	// Row 2: Time (seconds)
	GVL_HMI.aSolventAndTimesRows[2].Rinse1 := DWORD_TO_INT(TIME_TO_DWORD(GVL_Recipe.stCurrentRecipe.stSolventsTimes.aTime[1]) / 1000); // TIME in seconds
	GVL_HMI.aSolventAndTimesRows[2].Rinse2 := DWORD_TO_INT(TIME_TO_DWORD(GVL_Recipe.stCurrentRecipe.stSolventsTimes.aTime[2]) / 1000); // TIME in seconds
	GVL_HMI.aSolventAndTimesRows[2].Wash1  := DWORD_TO_INT(TIME_TO_DWORD(GVL_Recipe.stCurrentRecipe.stSolventsTimes.aTime[3]) / 1000); // TIME in seconds
	GVL_HMI.aSolventAndTimesRows[2].Wash2  := DWORD_TO_INT(TIME_TO_DWORD(GVL_Recipe.stCurrentRecipe.stSolventsTimes.aTime[4]) / 1000); // TIME in seconds
	
	// Row 3: Velocity
	GVL_HMI.aSolventAndTimesRows[3].Rinse1 := GVL_Recipe.stCurrentRecipe.stSolventsTimes.aVelocity[1];
	GVL_HMI.aSolventAndTimesRows[3].Rinse2 := GVL_Recipe.stCurrentRecipe.stSolventsTimes.aVelocity[2];
	GVL_HMI.aSolventAndTimesRows[3].Wash1  := GVL_Recipe.stCurrentRecipe.stSolventsTimes.aVelocity[3];
	GVL_HMI.aSolventAndTimesRows[3].Wash2  := GVL_Recipe.stCurrentRecipe.stSolventsTimes.aVelocity[4];
	
	//Volumes Datagrid
	// 1:Rinse1, 2:Rinse2, 3:Wash1, 4:Wash2
    GVL_HMI.aVolumeRows[1].Rinse1 := GVL_Recipe.stCurrentRecipe.stVolumes.aT_IC_Volume[1];
    GVL_HMI.aVolumeRows[1].Rinse2 := GVL_Recipe.stCurrentRecipe.stVolumes.aT_IC_Volume[2];
    GVL_HMI.aVolumeRows[1].Wash1  := GVL_Recipe.stCurrentRecipe.stVolumes.aT_IC_Volume[3];
    GVL_HMI.aVolumeRows[1].Wash2  := GVL_Recipe.stCurrentRecipe.stVolumes.aT_IC_Volume[4];

    GVL_HMI.aVolumeRows[2].Rinse1 := GVL_Recipe.stCurrentRecipe.stVolumes.aS0_Volume[1];
    GVL_HMI.aVolumeRows[2].Rinse2 := GVL_Recipe.stCurrentRecipe.stVolumes.aS0_Volume[2];
    GVL_HMI.aVolumeRows[2].Wash1  := GVL_Recipe.stCurrentRecipe.stVolumes.aS0_Volume[3];
    GVL_HMI.aVolumeRows[2].Wash2  := GVL_Recipe.stCurrentRecipe.stVolumes.aS0_Volume[4];

    GVL_HMI.aVolumeRows[3].Rinse1 := GVL_Recipe.stCurrentRecipe.stVolumes.aS1_Volume[1];
    GVL_HMI.aVolumeRows[3].Rinse2 := GVL_Recipe.stCurrentRecipe.stVolumes.aS1_Volume[2];
   	GVL_HMI.aVolumeRows[3].Wash1  := GVL_Recipe.stCurrentRecipe.stVolumes.aS1_Volume[3];
    GVL_HMI.aVolumeRows[3].Wash2  := GVL_Recipe.stCurrentRecipe.stVolumes.aS1_Volume[4];
	
	GVL_HMI.aVolumeRows[4].Rinse1 := GVL_Recipe.stCurrentRecipe.stVolumes.aS2_Volume[1];
    GVL_HMI.aVolumeRows[4].Rinse2 := GVL_Recipe.stCurrentRecipe.stVolumes.aS2_Volume[2];
   	GVL_HMI.aVolumeRows[4].Wash1  := GVL_Recipe.stCurrentRecipe.stVolumes.aS2_Volume[3];
    GVL_HMI.aVolumeRows[4].Wash2  := GVL_Recipe.stCurrentRecipe.stVolumes.aS2_Volume[4];
	
	GVL_HMI.aVolumeRows[5].Rinse1 := GVL_Recipe.stCurrentRecipe.stVolumes.aS3_Volume[1];
    GVL_HMI.aVolumeRows[5].Rinse2 := GVL_Recipe.stCurrentRecipe.stVolumes.aS3_Volume[2];
   	GVL_HMI.aVolumeRows[5].Wash1  := GVL_Recipe.stCurrentRecipe.stVolumes.aS3_Volume[3];
    GVL_HMI.aVolumeRows[5].Wash2  := GVL_Recipe.stCurrentRecipe.stVolumes.aS3_Volume[4];
	
	GVL_HMI.aVolumeRows[6].Rinse1 := GVL_Recipe.stCurrentRecipe.stVolumes.aS4_Volume[1];
    GVL_HMI.aVolumeRows[6].Rinse2 := GVL_Recipe.stCurrentRecipe.stVolumes.aS4_Volume[2];
   	GVL_HMI.aVolumeRows[6].Wash1  := GVL_Recipe.stCurrentRecipe.stVolumes.aS4_Volume[3];
    GVL_HMI.aVolumeRows[6].Wash2  := GVL_Recipe.stCurrentRecipe.stVolumes.aS4_Volume[4];
	
	GVL_HMI.aVolumeRows[7].Rinse1 := GVL_Recipe.stCurrentRecipe.stVolumes.aS5_Volume[1];
    GVL_HMI.aVolumeRows[7].Rinse2 := GVL_Recipe.stCurrentRecipe.stVolumes.aS5_Volume[2];
   	GVL_HMI.aVolumeRows[7].Wash1  := GVL_Recipe.stCurrentRecipe.stVolumes.aS5_Volume[3];
    GVL_HMI.aVolumeRows[7].Wash2  := GVL_Recipe.stCurrentRecipe.stVolumes.aS5_Volume[4];
	
	GVL_HMI.aVolumeRows[8].Rinse1 := GVL_Recipe.stCurrentRecipe.stVolumes.aS6_Volume[1];
    GVL_HMI.aVolumeRows[8].Rinse2 := GVL_Recipe.stCurrentRecipe.stVolumes.aS6_Volume[2];
   	GVL_HMI.aVolumeRows[8].Wash1  := GVL_Recipe.stCurrentRecipe.stVolumes.aS6_Volume[3];
    GVL_HMI.aVolumeRows[8].Wash2  := GVL_Recipe.stCurrentRecipe.stVolumes.aS6_Volume[4];
	
	GVL_HMI.aVolumeRows[9].Rinse1 := GVL_Recipe.stCurrentRecipe.stVolumes.aS7_Volume[1];
    GVL_HMI.aVolumeRows[9].Rinse2 := GVL_Recipe.stCurrentRecipe.stVolumes.aS7_Volume[2];
   	GVL_HMI.aVolumeRows[9].Wash1  := GVL_Recipe.stCurrentRecipe.stVolumes.aS7_Volume[3];
    GVL_HMI.aVolumeRows[9].Wash2  := GVL_Recipe.stCurrentRecipe.stVolumes.aS7_Volume[4];

    GVL_HMI.aVolumeRows[10].Rinse1 := GVL_Recipe.stCurrentRecipe.stVolumes.aF_Volume[1];
    GVL_HMI.aVolumeRows[10].Rinse2 := GVL_Recipe.stCurrentRecipe.stVolumes.aF_Volume[2];
    GVL_HMI.aVolumeRows[10].Wash1  := GVL_Recipe.stCurrentRecipe.stVolumes.aF_Volume[3];
    GVL_HMI.aVolumeRows[10].Wash2  := GVL_Recipe.stCurrentRecipe.stVolumes.aF_Volume[4];
	
	//Other Params datagrid
	GVL_HMI.aOtherParamsRows[1].Value     := TIME_TO_DWORD(GVL_Recipe.stCurrentRecipe.stOtherParams.tSoakTime) / 1000.0; // Soak Time
	GVL_HMI.aOtherParamsRows[2].Value     := TIME_TO_DWORD(GVL_Recipe.stCurrentRecipe.stOtherParams.tAgitate1Time) / 1000.0; // Agitate 1 Time
	GVL_HMI.aOtherParamsRows[3].Value     := TIME_TO_DWORD(GVL_Recipe.stCurrentRecipe.stOtherParams.tAgitate2Time) / 1000.0; // Agitate 2 Time
	GVL_HMI.aOtherParamsRows[4].Value     := GVL_Recipe.stCurrentRecipe.stOtherParams.iVialsToFill; // Vials to Fill
	GVL_HMI.aOtherParamsRows[5].Value     := GVL_Recipe.stCurrentRecipe.stOtherParams.rVialPrimeVol; // Vial Prime Vol
	GVL_HMI.aOtherParamsRows[6].Value     := GVL_Recipe.stCurrentRecipe.stOtherParams.rVial1FillVol; // Vial 1 Fill Vol
	GVL_HMI.aOtherParamsRows[7].Value     := GVL_Recipe.stCurrentRecipe.stOtherParams.rVials2_4FillVol; // Vials 2-4 Fill Vol
	GVL_HMI.aOtherParamsRows[8].Value     := TIME_TO_DWORD(GVL_Recipe.stCurrentRecipe.stOtherParams.tAirDryTime) / 1000.0; // Air Dry Time
	
	iStep := 100;

90:
    fbFileClose(sNetId := '', hFile := hFile, bExecute := TRUE);
    iStep := 100;
	
100:
    bBusy := FALSE;
    bDone := NOT bError;
    IF NOT bExecute THEN
        iStep := 0;
    END_IF
END_CASE

END_FUNCTION_BLOCK

// ---- POUs/4. RecipeHandle/FB_ListRecipeFiles.TcPOU
// FB_ListRecipeFiles: Scans the recipe folder and fills GVL_Recipe.aAvailableFiles with metadata from JSON files
FUNCTION_BLOCK FB_ListRecipeFiles
VAR_INPUT
	bExecute : BOOL; // Start the file listing process
END_VAR
VAR_OUTPUT
	bBusy       : BOOL; // Indicates the block is busy
    bError      : BOOL; // Indicates an error occurred
    nErrId      : UDINT; // Error code if any
	bDone   	: BOOL;

END_VAR
VAR
	fbEnumFiles     : FB_EnumFindFileList;
    fbFileTime      : FB_FileTime64ToTzSpecificLocalTime;
    fbHeaderHandler : FB_RecipeHeaderHandler;

    aFindBuffer     : ARRAY[0..49] OF ST_FindFileEntry;
    nFoundFiles     : UDINT;
    iFileIndex      : INT;
    iStep           : INT;
    bExecutePrev    : BOOL;
    bStart          : BOOL;
    bHeaderHandlerReset : BOOL;
    bHeaderHandlerExecute : BOOL;
	
	i : INT;
	
END_VAR

bStart := NOT bExecutePrev AND bExecute;
bExecutePrev := bExecute;

IF NOT bExecute THEN
	bBusy := FALSE;
  	bDone := FALSE;
	bError := FALSE;
	nErrId := 0;
END_IF

CASE iStep OF

0:
    IF bStart THEN
        bBusy := TRUE;
        bDone := FALSE;
        bError := FALSE;
        nErrId := 0;
        iFileIndex := 0;
        bHeaderHandlerReset := FALSE;
        bHeaderHandlerExecute := FALSE;

        fbEnumFiles(
            sNetId := '',
            sPathName := 'C:/TwinCAT/Recipes/*.json',
            eCmd := eEnumCmd_First,
            pFindList := ADR(aFindBuffer),
            cbFindList := SIZEOF(aFindBuffer),
            bExecute := TRUE
        );

        iStep := 10;
    END_IF

10:
    fbEnumFiles(bExecute := FALSE);
    IF NOT fbEnumFiles.bBusy THEN
        IF fbEnumFiles.bError THEN
            bError := TRUE;
            nErrId := fbEnumFiles.nErrId;
            iStep := 100;
        ELSE
            nFoundFiles := fbEnumFiles.nFindFiles;
            IF nFoundFiles > 0 THEN
                iStep := 20;
            ELSE
                bDone := TRUE;
                iStep := 100;
            END_IF
        END_IF
    END_IF

// 20 - Processa arquivo iFileIndex
20:
    IF iFileIndex < TO_INT(nFoundFiles) AND iFileIndex <= 49 THEN
        // Preenche campos básicos do arquivo
        GVL_HMI.aAvailableFiles[iFileIndex].sFileName := aFindBuffer[iFileIndex].sFileName;
        fbFileTime(
            in := FILETIME_TO_FILETIME64(aFindBuffer[iFileIndex].lastWriteTime),
            tzInfo := WEST_EUROPE_TZI
        );
        GVL_HMI.aAvailableFiles[iFileIndex].dtLastModified := FILETIME64_TO_DT(fbFileTime.out);

        // Vai para o step de reset do FB_HeaderHandler
        iStep := 21;
    ELSE
        bDone := TRUE;
        iStep := 100;
    END_IF

// 21 - Reset do FB_HeaderHandler (chamada com bExecute := FALSE por um ciclo)
21:
    fbHeaderHandler(bExecute := FALSE);
    IF NOT fbHeaderHandler.bBusy AND NOT fbHeaderHandler.bDone THEN
        iStep := 22;
    END_IF

// 22 - Chama o FB_HeaderHandler para ler o header do arquivo atual
22:
    fbHeaderHandler(
        sFileName := CONCAT('C:/TwinCAT/Recipes/', aFindBuffer[iFileIndex].sFileName),
        iTargetIndex := iFileIndex,
        bExecute := TRUE
    );
    IF NOT fbHeaderHandler.bBusy THEN
        IF fbHeaderHandler.bError THEN
            bError := TRUE;
            nErrId := fbHeaderHandler.nErrId;
            iStep := 100;
        ELSIF fbHeaderHandler.bDone THEN
            iStep := 23;
        END_IF
    END_IF

23: // Dummy step — aguarda 1 ciclo antes de liberar novo arquivo
    fbHeaderHandler(bExecute := FALSE);
    iFileIndex := iFileIndex + 1;
    iStep := 20;

100:
    bBusy := FALSE;
    IF NOT bExecute THEN
        iStep := 0;
    END_IF
END_CASE

END_FUNCTION_BLOCK

// ---- POUs/4. RecipeHandle/FB_RecipeHeaderHandler.TcPOU
// FB_RecipeHeaderHandler: Extracts metadata from a recipe JSON file and fills one entry in GVL_Recipe.aAvailableFiles
FUNCTION_BLOCK FB_RecipeHeaderHandler
VAR_INPUT
	sFileName       : STRING(255);
    iTargetIndex    : INT; // Index to write into array GVL_Recipe.aAvailableFiles
    bExecute        : BOOL;
END_VAR
VAR_OUTPUT
	bBusy  : BOOL;
    bError : BOOL;
    bDone  : BOOL;
    nErrId : UDINT;
END_VAR
VAR
	iStep         : INT;
    hFile         : UINT;
    sBuffer       : STRING(8192);
    fbFileOpen    : FB_FileOpen;
    fbFileRead    : FB_FileRead;
    fbFileClose   : FB_FileClose;
    fbJson        : FB_JsonDomParser;
    jsonDoc       : SJsonValue;
    jsonProp      : SJsonValue;
	nBytesRead    : UDINT;
	bExecutePrev  : BOOL; 
    bStart        : BOOL;
	bWait1Cycle	  : BOOL := FALSE;
	iCount		  : UINT := 0;
	iDummyTimer	  : INT := 0;
END_VAR

bStart := bExecute AND NOT bExecutePrev;
bExecutePrev := bExecute;

IF NOT bExecute THEN
	bBusy := FALSE;
    bDone := FALSE;
    bError := FALSE;

	sBuffer := '';
	jsonDoc := 0;
	jsonProp := 0;
	hFile := 0;
	bExecutePrev := FALSE;	
END_IF

CASE iStep OF

0:
     IF bExecute AND NOT bBusy THEN
        bBusy := TRUE;
        bDone := FALSE;
        bError := FALSE;
        nErrId := 0;
        iCount := 0;
        // Reset interno total
        sBuffer := '';
        jsonDoc := 0;
        jsonProp := 0;
        hFile := 0;
        iStep := 5;
    END_IF
	
5:
	fbFileOpen(
            sNetId := '',
            sPathName := sFileName,
            nMode := FOPEN_MODEREAD OR FOPEN_MODETEXT,
            bExecute := TRUE,
			hFile => hFile
	);
	IF NOT fbFileOpen.bBusy AND NOT fbFileOpen.bError THEN
		iStep := 10;
	END_IF

10:
    fbFileOpen(
        sNetId := '',
        sPathName := sFileName,
        nMode := FOPEN_MODEREAD OR FOPEN_MODETEXT,
        bExecute := FALSE
    );
    IF NOT fbFileOpen.bBusy THEN
        IF fbFileOpen.bError THEN
            bError := TRUE;
            nErrId := fbFileOpen.nErrId;
            iStep := 100;
        ELSE
            hFile := fbFileOpen.hFile;
            fbFileRead(
                sNetId := '',
                hFile := hFile,
                pReadBuff := ADR(sBuffer),
                cbReadLen := SIZEOF(sBuffer),
                bExecute := TRUE
            );
            iStep := 20;
        END_IF
    END_IF

20:
    fbFileRead(
        sNetId := '',
        hFile := hFile,
        pReadBuff := ADR(sBuffer),
        cbReadLen := SIZEOF(sBuffer),
        bExecute := FALSE,
        cbRead => nBytesRead 
    );
    IF NOT fbFileRead.bBusy THEN
        IF fbFileRead.bError THEN
            bError := TRUE;
            nErrId := fbFileRead.nErrId;
            iStep := 100;
        ELSE
            // Clear the buffer
            IF nBytesRead < SIZEOF(sBuffer) THEN
    			sBuffer[nBytesRead] := 0; 
			END_IF

            fbFileClose(
                sNetId := '',
                hFile := hFile,
                bExecute := TRUE
            );
            iStep := 30;
        END_IF
    END_IF


30:
    fbFileClose(
        sNetId := '',
        hFile := hFile,
        bExecute := FALSE
    );
    IF NOT fbFileClose.bBusy THEN
        IF fbFileClose.bError THEN
            bError := TRUE;
            nErrId := fbFileClose.nErrId;
            iStep := 100;
        ELSE
            iStep := 31;
        END_IF
    END_IF

31: // Dummy step: espera um ciclo para garantir flush/GC do Windows
	fbFileClose( sNetId := '', hFile := hFile, bExecute := FALSE );
	hFile := 0; // <- ZERA handle explicitamente!
    iDummyTimer := iDummyTimer + 1;
    IF iDummyTimer > 1 THEN
        iDummyTimer := 0;
        iStep := 32; // Continua
    END_IF

32: 
	jsonDoc := fbJson.ParseDocument(sBuffer);
	IF jsonDoc = 0 THEN
		iStep := 35;
	ELSE
		iStep := 40;
	END_IF

35:
	IF iCount > 10 THEN 
		bError := TRUE;
		nErrId := 16#F1000001; // Custom error code for invalid JSON
		iStep := 100;
	ELSE
		jsonDoc := 0;
		jsonProp := 0;
		sBuffer := '';
		iCount := iCount + 1;
		iStep := 0;
	END_IF
	
39:
	IF bWait1Cycle THEN
		iStep := 40;
	END_IF 
	IF NOT bWait1Cycle THEN
		bWait1Cycle := TRUE;
	END_IF

40:
	bWait1Cycle := FALSE;
	
	// Extract sMethodName
	jsonProp := fbJson.FindMemberPath(jsonDoc, 'stInfo/sMethodName');
	GVL_HMI.aAvailableFiles[iTargetIndex].sMethodName := fbJson.GetString(jsonProp);
	
    // Extract sCreatedBy
	jsonProp := fbJson.FindMemberPath(jsonDoc, 'stInfo/sCreatedBy');
	GVL_HMI.aAvailableFiles[iTargetIndex].sCreatedBy := fbJson.GetString(jsonProp);

    // Extract dCreationDate
    jsonProp := fbJson.FindMemberPath(jsonDoc, 'stInfo/dCreationDate');
    GVL_HMI.aAvailableFiles[iTargetIndex].dCreationDate := STRING_TO_DATE(fbJson.GetString(jsonProp));

    // Extract iRevision
    jsonProp := fbJson.FindMemberPath(jsonDoc, 'stInfo/iRevision');
    GVL_HMI.aAvailableFiles[iTargetIndex].iRevision := TO_INT(fbJson.GetInt(jsonProp));

    iStep := 100;

100:
    bBusy := FALSE;
    bDone := TRUE;
	bExecutePrev := FALSE;
	icount := 0;
    IF NOT bExecute THEN
        iStep := 0;
    END_IF

END_CASE

END_FUNCTION_BLOCK

// ---- POUs/4. RecipeHandle/FB_DeleteRecipe.TcPOU
FUNCTION_BLOCK FB_DeleteRecipe
VAR_INPUT
    bExecute      : BOOL; // Trigger (rising edge)
    stFileInfo    : ST_RecipeFileInfo; // Info da receita a deletar
END_VAR
VAR_OUTPUT
    bBusy   : BOOL;
    bDone   : BOOL;
    bError  : BOOL;
    nErrId  : UDINT;
END_VAR
VAR
    iStep         : INT;
    fbFileRename  : FB_FileRename;
    sOldPath      : STRING(256);
    sNewPath      : STRING(256);
END_VAR

CASE iStep OF
0:
    IF bExecute THEN
        bBusy := TRUE; bDone := FALSE; bError := FALSE; nErrId := 0;
        // Monta caminhos
        sOldPath := CONCAT('C:/TwinCAT/Recipes/', CONCAT(stFileInfo.sFileName, '.json'));
        sNewPath := CONCAT('C:/TwinCAT/Recipes/_deleted/', CONCAT(stFileInfo.sFileName, '.json'));

        // Executa rename/move
        fbFileRename(
            sNetId := '',
            sOldName := sOldPath,
            sNewName := sNewPath,
            bExecute := TRUE
        );
        iStep := 10;
    END_IF

10:
    fbFileRename(bExecute := FALSE);
    IF NOT fbFileRename.bBusy THEN
        IF fbFileRename.bError THEN
            bError := TRUE;
            nErrId := fbFileRename.nErrId;
            bDone := FALSE;
            bBusy := FALSE;
            iStep := 100;
        ELSE
            bDone := TRUE;
            bBusy := FALSE;
            bError := FALSE;
            iStep := 100;
        END_IF
    END_IF

100:
    IF NOT bExecute THEN
        iStep := 0;
        bDone := FALSE;
        bBusy := FALSE;
        bError := FALSE;
    END_IF
END_CASE

END_FUNCTION_BLOCK

// ---- POUs/4. RecipeHandle/FB_SaveRecipe.TcPOU
FUNCTION_BLOCK FB_SaveRecipe
VAR_INPUT
    bExecute : BOOL;           // Trigger to start the save operation (level-sensitive)
    sUser    : STRING(64);     // Operator/user name to stamp into the recipe header
END_VAR
VAR_OUTPUT
    bDone    : BOOL;           // TRUE when the save operation completes successfully
    bBusy    : BOOL;           // TRUE while the state machine is running
    bError   : BOOL;           // TRUE if an error occurs in any file operation
    nErrId   : UDINT;          // Error code from file function blocks
END_VAR
VAR
    // --- State machine and helpers ---
    iStep         : INT;                       // Current state
    fbJson        : FB_JsonDomParser;          // JSON DOM builder
    sJsonBuffer   : STRING(8192);              // Output buffer for JSON serialization
    sFileName     : STRING(256);               // New file full path
    sOldFile      : STRING(256);               // Previous revision file path
    sOldBackup    : STRING(256);               // Backup path for previous revision
    sTempStr      : STRING(64);                // Temporary string for conversions
    iTempNumb     : DINT;                      // Temporary integer for conversions

    // --- File handling FBs ---
    fbFileOpen    : FB_FileOpen;
    fbFileWrite   : FB_FileWrite;
    fbFileClose   : FB_FileClose;
    fbFileRename  : FB_FileRename;
    nBytesToWrite : UDINT;                     // Number of bytes to write (excludes trailing 0)
    hFile         : UINT;                      // File handle

    // --- Date/Time stamping ---
    fbLocalSystemTime : FB_LocalSystemTime;    // Reads IPC local time
    sDate             : STRING(12);            // "D#YYYY-MM-DD" to convert with STRING_TO_DATE
    stLocalSystemTime : TIMESTRUCT;            // System time structure
    tzID              : E_TimeZoneID := eTimeZoneID_Invalid; // (Unused here; placeholder)

    // --- JSON nodes ---
    jsonRoot, objStInfo, objSolventsTimes, objVolumes, objOtherParams : SJsonValue;
    arrVal : SJsonValue;
    i : INT;

    // --- One-shot guards within a single execution ---
    bRevisionDone       : BOOL := FALSE;       // Ensures revision logic runs once per execution
    bGetCurrentDateDone : BOOL := FALSE;       // Ensures date capture runs once per execution
	
END_VAR

// === STATE MACHINE ===
CASE iStep OF

// -------------------------------------------------------------
// 0: Idle / Entry. Wait for bExecute to start the save routine.
// -------------------------------------------------------------
0:
    IF bExecute THEN
        // Initialize outputs and flags
        bBusy  := TRUE;
        bDone  := FALSE;
        bError := FALSE;
        nErrId := 0;

        // --- Revision handling (run once) ---
        // If "New Recipe" button was used, start at revision 0.
        // Otherwise, increment the existing revision by 1.
        IF NOT bRevisionDone THEN
            IF GVL_HMI.bNewRecipeButton THEN
                GVL_Recipe.stCurrentRecipe.stInfo.iRevision := 0;
                bRevisionDone := TRUE;
            ELSE
                GVL_Recipe.stCurrentRecipe.stInfo.iRevision := GVL_Recipe.stCurrentRecipe.stInfo.iRevision + 1;
                bRevisionDone := TRUE;
            END_IF
        END_IF

        // --- Get local system date/time (run until valid once) ---
        // This block enables the clock reader and, when valid, produces TIMESTRUCT.
        fbLocalSystemTime(bEnable := TRUE, dwCycle := 5);
        IF fbLocalSystemTime.bValid THEN
            stLocalSystemTime := fbLocalSystemTime.systemTime;

            // Build date string "D#YYYY-MM-DD" required by STRING_TO_DATE
            sDate := CONCAT('D#', INT_TO_STRING(stLocalSystemTime.wYear));
            sDate := CONCAT(sDate, '-');
            sDate := CONCAT(sDate, INT_TO_STRING(stLocalSystemTime.wMonth));
            sDate := CONCAT(sDate, '-');
            sDate := CONCAT(sDate, INT_TO_STRING(stLocalSystemTime.wDay));

            // Persist date into recipe header (DATE type)
            GVL_Recipe.stCurrentRecipe.stInfo.dCreationDate := STRING_TO_DATE(sDate);
            bGetCurrentDateDone := TRUE;
        END_IF

        // Only proceed once date/time was captured
        IF bGetCurrentDateDone THEN

            // Stamp the creator name
            GVL_Recipe.stCurrentRecipe.stInfo.sCreatedBy := sUser;

            // --- Compose file names ---
            // New file: .../<Method>_<User>_rev<Revision>.json
            sFileName := CONCAT('C:/TwinCAT/Recipes/',
                CONCAT(GVL_Recipe.stCurrentRecipe.stInfo.sMethodName, CONCAT('_',
                CONCAT(sUser, CONCAT('_rev', CONCAT(DINT_TO_STRING(GVL_Recipe.stCurrentRecipe.stInfo.iRevision), '.json')))))
            );

            // Previous file (revision-1) for backup (no fatal error if it doesn't exist)
            sOldFile := CONCAT('C:/TwinCAT/Recipes/',
                CONCAT(GVL_Recipe.stCurrentRecipe.stInfo.sMethodName, CONCAT('_',
                CONCAT(sUser, CONCAT('_rev', CONCAT(DINT_TO_STRING(GVL_Recipe.stCurrentRecipe.stInfo.iRevision - 1), '.json')))))
            );

            // Backup path for the previous file
            sOldBackup := CONCAT('C:/TwinCAT/Recipes/_old/',
                CONCAT(GVL_Recipe.stCurrentRecipe.stInfo.sMethodName, CONCAT('_',
                CONCAT(sUser, CONCAT('_rev', CONCAT(DINT_TO_STRING(GVL_Recipe.stCurrentRecipe.stInfo.iRevision - 1), '.json')))))
            );

            // --- Build JSON document ---
            jsonRoot := fbJson.NewDocument();

            // Header: stInfo
            objStInfo := fbJson.AddObjectMember(jsonRoot, 'stInfo');
            fbJson.AddStringMember(objStInfo, 'sMethodName', GVL_Recipe.stCurrentRecipe.stInfo.sMethodName);
            fbJson.AddIntMember   (objStInfo, 'iRevision',   GVL_Recipe.stCurrentRecipe.stInfo.iRevision);
            fbJson.AddStringMember(objStInfo, 'sCreatedBy',  GVL_Recipe.stCurrentRecipe.stInfo.sCreatedBy);
            sTempStr := DATE_TO_STRING(GVL_Recipe.stCurrentRecipe.stInfo.dCreationDate);
            fbJson.AddStringMember(objStInfo, 'dCreationDate', sTempStr);

            // stSolventsTimes
            objSolventsTimes := fbJson.AddObjectMember(jsonRoot, 'stSolventsTimes');

            // aSolventN[1..4] as integer array
            arrVal := fbJson.AddArrayMember(objSolventsTimes, 'aSolventN', 0);
            FOR i := 1 TO 4 DO
                fbJson.PushbackIntValue(arrVal, GVL_Recipe.stCurrentRecipe.stSolventsTimes.aSolventN[i]);
            END_FOR

            // aTime[1..4] as stringified TIME array (e.g., "T#10S")
            arrVal := fbJson.AddArrayMember(objSolventsTimes, 'aTime', 0);
            FOR i := 1 TO 4 DO
                sTempStr := TIME_TO_STRING(GVL_Recipe.stCurrentRecipe.stSolventsTimes.aTime[i]);
                fbJson.PushbackStringValue(arrVal, sTempStr);
            END_FOR

            // aVelocity[1..4] as integer array
            arrVal := fbJson.AddArrayMember(objSolventsTimes, 'aVelocity', 0);
            FOR i := 1 TO 4 DO
                fbJson.PushbackIntValue(arrVal, GVL_Recipe.stCurrentRecipe.stSolventsTimes.aVelocity[i]);
            END_FOR

            // stVolumes (multiple double arrays, each [1..4])
            objVolumes := fbJson.AddObjectMember(jsonRoot, 'stVolumes');

            arrVal := fbJson.AddArrayMember(objVolumes, 'aT_IC_Volume', 0);
            FOR i := 1 TO 4 DO fbJson.PushbackDoubleValue(arrVal, GVL_Recipe.stCurrentRecipe.stVolumes.aT_IC_Volume[i]); END_FOR

            arrVal := fbJson.AddArrayMember(objVolumes, 'aS0_Volume', 0);
            FOR i := 1 TO 4 DO fbJson.PushbackDoubleValue(arrVal, GVL_Recipe.stCurrentRecipe.stVolumes.aS0_Volume[i]); END_FOR

            arrVal := fbJson.AddArrayMember(objVolumes, 'aS1_Volume', 0);
            FOR i := 1 TO 4 DO fbJson.PushbackDoubleValue(arrVal, GVL_Recipe.stCurrentRecipe.stVolumes.aS1_Volume[i]); END_FOR

            arrVal := fbJson.AddArrayMember(objVolumes, 'aS2_Volume', 0);
            FOR i := 1 TO 4 DO fbJson.PushbackDoubleValue(arrVal, GVL_Recipe.stCurrentRecipe.stVolumes.aS2_Volume[i]); END_FOR

            arrVal := fbJson.AddArrayMember(objVolumes, 'aS3_Volume', 0);
            FOR i := 1 TO 4 DO fbJson.PushbackDoubleValue(arrVal, GVL_Recipe.stCurrentRecipe.stVolumes.aS3_Volume[i]); END_FOR

            arrVal := fbJson.AddArrayMember(objVolumes, 'aS4_Volume', 0);
            FOR i := 1 TO 4 DO fbJson.PushbackDoubleValue(arrVal, GVL_Recipe.stCurrentRecipe.stVolumes.aS4_Volume[i]); END_FOR

            arrVal := fbJson.AddArrayMember(objVolumes, 'aS5_Volume', 0);
            FOR i := 1 TO 4 DO fbJson.PushbackDoubleValue(arrVal, GVL_Recipe.stCurrentRecipe.stVolumes.aS5_Volume[i]); END_FOR

            arrVal := fbJson.AddArrayMember(objVolumes, 'aS6_Volume', 0);
            FOR i := 1 TO 4 DO fbJson.PushbackDoubleValue(arrVal, GVL_Recipe.stCurrentRecipe.stVolumes.aS6_Volume[i]); END_FOR

            arrVal := fbJson.AddArrayMember(objVolumes, 'aS7_Volume', 0);
            FOR i := 1 TO 4 DO fbJson.PushbackDoubleValue(arrVal, GVL_Recipe.stCurrentRecipe.stVolumes.aS7_Volume[i]); END_FOR

            arrVal := fbJson.AddArrayMember(objVolumes, 'aF_Volume', 0);
            FOR i := 1 TO 4 DO fbJson.PushbackDoubleValue(arrVal, GVL_Recipe.stCurrentRecipe.stVolumes.aF_Volume[i]); END_FOR

            // stOtherParams
            objOtherParams := fbJson.AddObjectMember(jsonRoot, 'stOtherParams');

            sTempStr := TIME_TO_STRING(GVL_Recipe.stCurrentRecipe.stOtherParams.tSoakTime);
            fbJson.AddStringMember(objOtherParams, 'tSoakTime', sTempStr);

            sTempStr := TIME_TO_STRING(GVL_Recipe.stCurrentRecipe.stOtherParams.tAgitate1Time);
            fbJson.AddStringMember(objOtherParams, 'tAgitate1Time', sTempStr);

            sTempStr := TIME_TO_STRING(GVL_Recipe.stCurrentRecipe.stOtherParams.tAgitate2Time);
            fbJson.AddStringMember(objOtherParams, 'tAgitate2Time', sTempStr);

            iTempNumb := TO_DINT(GVL_Recipe.stCurrentRecipe.stOtherParams.iVialsToFill);
            fbJson.AddIntMember(objOtherParams, 'iVialsToFill', iTempNumb);

            fbJson.AddDoubleMember(objOtherParams, 'rVialPrimeVol',   GVL_Recipe.stCurrentRecipe.stOtherParams.rVialPrimeVol);
            fbJson.AddDoubleMember(objOtherParams, 'rVial1FillVol',   GVL_Recipe.stCurrentRecipe.stOtherParams.rVial1FillVol);
            fbJson.AddDoubleMember(objOtherParams, 'rVials2_4FillVol', GVL_Recipe.stCurrentRecipe.stOtherParams.rVials2_4FillVol);

            sTempStr := TIME_TO_STRING(GVL_Recipe.stCurrentRecipe.stOtherParams.tAirDryTime);
            fbJson.AddStringMember(objOtherParams, 'tAirDryTime', sTempStr);

            // Serialize to buffer (also useful to precompute length)
            fbJson.CopyDocument(sJsonBuffer, SIZEOF(sJsonBuffer));

            // Ensure any previous rename FB is idle before proceeding
            fbFileRename(bExecute := FALSE);

            // Next step: try moving the old file to backup
            iStep := 5;
        END_IF
    END_IF

// -------------------------------------------------------------
// 5: Move old file to _old backup (non-fatal if not present).
//    Proceeds regardless of success; we don't block new save.
// -------------------------------------------------------------
5:
    fbFileRename(
        sNetId   := '',
        sOldName := sOldFile,
        sNewName := sOldBackup,
        bExecute := TRUE
    );

    // Make sure open FB is idle before reusing it later
    fbFileOpen(bExecute := FALSE);

    IF NOT fbFileRename.bBusy THEN
        // Ignore fbFileRename.bError intentionally: absence is acceptable
        iStep := 10;
    END_IF

// -------------------------------------------------------------
// 10: Create/open the new file for text write.
// -------------------------------------------------------------
10:
    fbFileOpen(
        sNetId    := '',
        sPathName := sFileName,
        nMode     := FOPEN_MODEWRITE OR FOPEN_MODETEXT, // Overwrite text file
        bExecute  := TRUE
    );

    // Keep write FB idle until we have a valid handle
    fbFileWrite(bExecute := FALSE);

    IF NOT fbFileOpen.bBusy THEN
        IF fbFileOpen.bError THEN
            bError := TRUE;
            nErrId := fbFileOpen.nErrId;
            iStep  := 100; // Go to end; wait for bExecute to drop
        ELSE
            hFile := fbFileOpen.hFile; // Store file handle
            iStep := 20;               // Proceed to write
        END_IF
    END_IF

// -------------------------------------------------------------
// 20: Write the serialized JSON buffer to disk.
// -------------------------------------------------------------
20:
    // Refresh serialized content and compute exact byte count (without trailing #0)
    nBytesToWrite := fbJson.CopyDocument(sJsonBuffer, SIZEOF(sJsonBuffer));
    IF nBytesToWrite > 0 THEN
        nBytesToWrite := nBytesToWrite - 1; // Exclude terminating null
    END_IF

    fbFileWrite(
        sNetId     := '',
        hFile      := hFile,
        pWriteBuff := ADR(sJsonBuffer),
        cbWriteLen := nBytesToWrite,
        bExecute   := TRUE
    );

    // Prepare close FB (idle for now)
    fbFileClose(bExecute := FALSE);

    IF NOT fbFileWrite.bBusy THEN
        IF fbFileWrite.bError THEN
            bError := TRUE;
            nErrId := fbFileWrite.nErrId;
            iStep  := 100; // Error path
        ELSE
            iStep := 30;   // Proceed to close
        END_IF
    END_IF

// -------------------------------------------------------------
// 30: Close the file, finalize flags, and finish.
// -------------------------------------------------------------
30:
    fbFileClose(
        sNetId   := '',
        hFile    := hFile,
        bExecute := TRUE
    );

    IF NOT fbFileClose.bBusy THEN
        IF fbFileClose.bError THEN
            bError := TRUE;
            nErrId := fbFileClose.nErrId;
        END_IF

        // Reset one-shot flags for a clean next cycle
        bGetCurrentDateDone := FALSE;
        GVL_HMI.bNewRecipeButton := FALSE;
        bRevisionDone := FALSE;

        // Mark completion
        bDone := TRUE;
        bBusy := FALSE;

        // Go to final state; wait for bExecute to drop
        iStep := 100;
    END_IF

// -------------------------------------------------------------
// 100: Final/hold state. Wait for bExecute to go FALSE to reset.
// -------------------------------------------------------------
100:
    IF NOT bExecute THEN
        // Reset to idle
        iStep := 0;

        // Clear guards and outputs to be ready for next run
        bRevisionDone       := FALSE;
        bGetCurrentDateDone := FALSE;
        bDone  := FALSE;
        bBusy  := FALSE;
        // bError/nErrId are intentionally kept until next run starts
    END_IF

END_CASE

END_FUNCTION_BLOCK

// ---- POUs/MARCO/DB/DB_Edit_Method.TcPOU
PROGRAM DB_Edit_Method
VAR
	state: INT;
	timer: ton;
	timer2: ton;
END_VAR

VAR_INPUT
	start: BOOL;
END_VAR

timer();
timer2();

CASE state OF
	
0:
	IF start THEN
		DB_Query.state:= E_DB_QUERY_STATE.INSERT_NEW_METHOD;
		timer(in:=TRUE, pt:=T#1S);
		state:= 5;
	ELSE
		state:= 0;
	END_IF

5:
	IF NOT DB_Query.FB_Insert.bBusy AND timer.Q THEN
		DB_Query.state:= E_DB_QUERY_STATE.SELECT_LAST_METHOD_ID;
		timer(in:=FALSE);
		timer2(in:= TRUE, pt:= T#1S);
		state:= 10; 
	ELSE
		state:= 5;
	END_IF

10:

	IF NOT DB_Query.FB_SelectArray.bBusy AND timer2.Q THEN
		timer2(in:=FALSE);
		
		GVL_DB.astVolData[1].pump := '1';
		GVL_DB.astVolData[1].stage := 'T/IC';
		GVL_DB.astVolData[1].rinse1 := REAL_TO_STRING(GVL_Recipe.stCurrentRecipe.stVolumes.aT_IC_Volume[1]);
		GVL_DB.astVolData[1].rinse2 := REAL_TO_STRING(GVL_Recipe.stCurrentRecipe.stVolumes.aT_IC_Volume[2]);
		GVL_DB.astVolData[1].wash1 := REAL_TO_STRING(GVL_Recipe.stCurrentRecipe.stVolumes.aT_IC_Volume[3]);
		GVL_DB.astVolData[1].wash2 := REAL_TO_STRING(GVL_Recipe.stCurrentRecipe.stVolumes.aT_IC_Volume[4]);
		GVL_DB.astVolData[2].pump := '2';
		GVL_DB.astVolData[2].stage := 'S0';
		GVL_DB.astVolData[2].rinse1 := REAL_TO_STRING(GVL_Recipe.stCurrentRecipe.stVolumes.aS0_Volume[1]);
		GVL_DB.astVolData[2].rinse2 := REAL_TO_STRING(GVL_Recipe.stCurrentRecipe.stVolumes.aS0_Volume[2]);
		GVL_DB.astVolData[2].wash1 := REAL_TO_STRING(GVL_Recipe.stCurrentRecipe.stVolumes.aS0_Volume[3]);
		GVL_DB.astVolData[2].wash2 := REAL_TO_STRING(GVL_Recipe.stCurrentRecipe.stVolumes.aS0_Volume[4]);
		GVL_DB.astVolData[3].pump := '3';
		GVL_DB.astVolData[3].stage := 'S1';
		GVL_DB.astVolData[3].rinse1 := REAL_TO_STRING(GVL_Recipe.stCurrentRecipe.stVolumes.aS1_Volume[1]);
		GVL_DB.astVolData[3].rinse2 := REAL_TO_STRING(GVL_Recipe.stCurrentRecipe.stVolumes.aS1_Volume[2]);
		GVL_DB.astVolData[3].wash1 := REAL_TO_STRING(GVL_Recipe.stCurrentRecipe.stVolumes.aS1_Volume[3]);
		GVL_DB.astVolData[3].wash2 := REAL_TO_STRING(GVL_Recipe.stCurrentRecipe.stVolumes.aS1_Volume[4]);
		GVL_DB.astVolData[4].pump := '4';
		GVL_DB.astVolData[4].stage := 'S2';
		GVL_DB.astVolData[4].rinse1 := REAL_TO_STRING(GVL_Recipe.stCurrentRecipe.stVolumes.aS2_Volume[1]);
		GVL_DB.astVolData[4].rinse2 := REAL_TO_STRING(GVL_Recipe.stCurrentRecipe.stVolumes.aS2_Volume[2]);
		GVL_DB.astVolData[4].wash1 := REAL_TO_STRING(GVL_Recipe.stCurrentRecipe.stVolumes.aS2_Volume[3]);
		GVL_DB.astVolData[4].wash2 := REAL_TO_STRING(GVL_Recipe.stCurrentRecipe.stVolumes.aS2_Volume[4]);
		GVL_DB.astVolData[5].pump := '5';
		GVL_DB.astVolData[5].stage := 'S3';
		GVL_DB.astVolData[5].rinse1 := REAL_TO_STRING(GVL_Recipe.stCurrentRecipe.stVolumes.aS3_Volume[1]);
		GVL_DB.astVolData[5].rinse2 := REAL_TO_STRING(GVL_Recipe.stCurrentRecipe.stVolumes.aS3_Volume[2]);
		GVL_DB.astVolData[5].wash1 := REAL_TO_STRING(GVL_Recipe.stCurrentRecipe.stVolumes.aS3_Volume[3]);
		GVL_DB.astVolData[5].wash2 := REAL_TO_STRING(GVL_Recipe.stCurrentRecipe.stVolumes.aS3_Volume[4]);
		GVL_DB.astVolData[6].pump := '6';
		GVL_DB.astVolData[6].stage := 'S4';
		GVL_DB.astVolData[6].rinse1 := REAL_TO_STRING(GVL_Recipe.stCurrentRecipe.stVolumes.aS4_Volume[1]);
		GVL_DB.astVolData[6].rinse2 := REAL_TO_STRING(GVL_Recipe.stCurrentRecipe.stVolumes.aS4_Volume[2]);
		GVL_DB.astVolData[6].wash1 := REAL_TO_STRING(GVL_Recipe.stCurrentRecipe.stVolumes.aS4_Volume[3]);
		GVL_DB.astVolData[6].wash2 := REAL_TO_STRING(GVL_Recipe.stCurrentRecipe.stVolumes.aS4_Volume[4]);
		GVL_DB.astVolData[7].pump := '7';
		GVL_DB.astVolData[7].stage := 'S5';
		GVL_DB.astVolData[7].rinse1 := REAL_TO_STRING(GVL_Recipe.stCurrentRecipe.stVolumes.aS5_Volume[1]);
		GVL_DB.astVolData[7].rinse2 := REAL_TO_STRING(GVL_Recipe.stCurrentRecipe.stVolumes.aS5_Volume[2]);
		GVL_DB.astVolData[7].wash1 := REAL_TO_STRING(GVL_Recipe.stCurrentRecipe.stVolumes.aS5_Volume[3]);
		GVL_DB.astVolData[7].wash2 := REAL_TO_STRING(GVL_Recipe.stCurrentRecipe.stVolumes.aS5_Volume[4]);
		GVL_DB.astVolData[8].pump := '8';
		GVL_DB.astVolData[8].stage := 'S6';
		GVL_DB.astVolData[8].rinse1 := REAL_TO_STRING(GVL_Recipe.stCurrentRecipe.stVolumes.aS6_Volume[1]);
		GVL_DB.astVolData[8].rinse2 := REAL_TO_STRING(GVL_Recipe.stCurrentRecipe.stVolumes.aS6_Volume[2]);
		GVL_DB.astVolData[8].wash1 := REAL_TO_STRING(GVL_Recipe.stCurrentRecipe.stVolumes.aS6_Volume[3]);
		GVL_DB.astVolData[8].wash2 := REAL_TO_STRING(GVL_Recipe.stCurrentRecipe.stVolumes.aS6_Volume[4]);
		GVL_DB.astVolData[9].pump := '9';
		GVL_DB.astVolData[9].stage := 'S7';
		GVL_DB.astVolData[9].rinse1 := REAL_TO_STRING(GVL_Recipe.stCurrentRecipe.stVolumes.aS7_Volume[1]);
		GVL_DB.astVolData[9].rinse2 := REAL_TO_STRING(GVL_Recipe.stCurrentRecipe.stVolumes.aS7_Volume[2]);
		GVL_DB.astVolData[9].wash1 := REAL_TO_STRING(GVL_Recipe.stCurrentRecipe.stVolumes.aS7_Volume[3]);
		GVL_DB.astVolData[9].wash2 := REAL_TO_STRING(GVL_Recipe.stCurrentRecipe.stVolumes.aS7_Volume[4]);
		GVL_DB.astVolData[10].pump := '10';
		GVL_DB.astVolData[10].stage := 'F';
		GVL_DB.astVolData[10].rinse1 := REAL_TO_STRING(GVL_Recipe.stCurrentRecipe.stVolumes.aF_Volume[1]);
		GVL_DB.astVolData[10].rinse2 := REAL_TO_STRING(GVL_Recipe.stCurrentRecipe.stVolumes.aF_Volume[2]);
		GVL_DB.astVolData[10].wash1 := REAL_TO_STRING(GVL_Recipe.stCurrentRecipe.stVolumes.aF_Volume[3]);
		GVL_DB.astVolData[10].wash2 := REAL_TO_STRING(GVL_Recipe.stCurrentRecipe.stVolumes.aF_Volume[4]);
		
		DB_Query.j := 1;
		state:= 20;
	ELSE
		state:= 10;
	END_IF
	
20:

	IF DB_Query.j <= 10 THEN
		DB_Query.state := E_DB_QUERY_STATE.INSERT_VOLUME_DATA;
		timer(in:=TRUE, pt:=T#2S);
		state:= 30;
	ELSIF DB_Query.j >10 THEN
		timer(in:=TRUE, pt:=T#1S);
		GVL_HMI.bRecipeSaveDone := TRUE;
		state:= 40;
	ELSE
		state:= 20;
	END_IF	

30:

	IF NOT DB_Query.FB_Insert.bBusy AND timer.Q THEN
		timer(in:=FALSE);
		DB_Query.j := DB_Query.j + 1;
		state:= 20;
	ELSE
		state:= 30;
	END_IF
	
40:

	IF NOT DB_Query.FB_Insert.bBusy AND timer.Q THEN
		IF NOT GVL_HMI.bNewRecipeButton THEN
			DB_Query.state := E_DB_QUERY_STATE.UPDATE_DEACTV_METHOD;
		END_IF
		timer(in:=FALSE);
		start:= FALSE;
		PRG_RecipeManager.bDatagridToRecipeDone := TRUE;
		GVL_HMI.bRecipeSaveDone := FALSE;
		state:= 0;
	ELSE
		state:= 40;
	END_IF
	
END_CASE

END_PROGRAM

// ---- POUs/Utilities/PRG_UserManagementHistory.TcPOU
PROGRAM PRG_UserManagementHistory
VAR
END_VAR

IF GVL_HMI.stUserMgmtHistoryEvent.bExecute 
AND DB_Query.state = E_DB_QUERY_STATE.IDLE_STATE THEN

    GVL_HMI.stUserMgmtHistoryEvent.bBusy := TRUE;
    GVL_HMI.stUserMgmtHistoryEvent.bDone := FALSE;
    GVL_HMI.stUserMgmtHistoryEvent.bError := FALSE;
    GVL_HMI.stUserMgmtHistoryEvent.sErrorText := '';

    DB_Query.state := E_DB_QUERY_STATE.INSERT_USER_MGMT_HISTORY;

END_IF

END_PROGRAM

// ---- POUs/MARCO/DB/DB_Load_SysParameters.TcPOU
PROGRAM DB_Load_SysParameters
VAR_INPUT
    bExecute : BOOL;
    bReset   : BOOL;
END_VAR

VAR_OUTPUT
    bBusy    : BOOL;
    bDone    : BOOL;
    bError   : BOOL;
    nErrorId : UDINT;
    nState   : INT;
END_VAR

VAR
   	state         : INT := 0;
    rExecute      : R_TRIG;
    tonTimeout    : TON;
    tTimeout      : TIME := T#10S;

    bQueryStarted : BOOL;
    bDbBusySeen   : BOOL;
END_VAR

rExecute(CLK := bExecute);

nState := state;

IF bReset THEN
    state := 0;
    bBusy := FALSE;
    bDone := FALSE;
    bError := FALSE;
    nErrorId := 0;
    bQueryStarted := FALSE;
    tonTimeout(IN := FALSE);
    RETURN;
END_IF


CASE state OF

    0: // IDLE
        bBusy := FALSE;
        
        IF NOT bDone THEN
            bError := FALSE;
            nErrorId := 0;
        END_IF

        tonTimeout(IN := FALSE);
        bQueryStarted := FALSE;

        IF rExecute.Q THEN
            bBusy := TRUE;
            bDone := FALSE;
            bError := FALSE;
            nErrorId := 0;
            state := 10;
        END_IF


    10: // REQUEST_LAST_SYSTEM_ID
		bBusy := TRUE;
	
		IF NOT bQueryStarted THEN
			DB_Query.state := E_DB_QUERY_STATE.SELECT_LAST_SYSTEM_ID;
			bQueryStarted := TRUE;
			bDbBusySeen := FALSE;
			tonTimeout(IN := TRUE, PT := tTimeout);
		END_IF
	
		tonTimeout(IN := TRUE, PT := tTimeout);
	
		IF DB_Query.FB_SelectArray.bBusy THEN
			bDbBusySeen := TRUE;
		END_IF
	
		IF bDbBusySeen AND NOT DB_Query.FB_SelectArray.bBusy THEN
			tonTimeout(IN := FALSE);
			bQueryStarted := FALSE;
			bDbBusySeen := FALSE;
			state := 20;
	
		ELSIF tonTimeout.Q THEN
			tonTimeout(IN := FALSE);
			bQueryStarted := FALSE;
			bDbBusySeen := FALSE;
			state := 900;
			nErrorId := 1001;
		END_IF


    20: // APPLY_SYSTEM_PARAMETERS
        GVL_Settings.sysRevNumber                                      := GVL_DB.stSysParameters.sysRevisionNo;
        GVL_Settings.sLastSysSettingsChangedBy                         := GVL_DB.stSysParameters.createdBy;
        GVL_Settings.sLastSysSettingsChangedOn                         := GVL_DB.stSysParameters.createdDate;

        GVL_Settings.stCalibParameters.rAcceptanceCriteria             := STRING_TO_LREAL(GVL_DB.stSysParameters.cal_AcceptanceCriteria);
        GVL_Settings.stCalibParameters.iAllowableFailures              := STRING_TO_USINT(GVL_DB.stSysParameters.cal_AllowableFail);
        GVL_Settings.stCalibParameters.iReplicatesSetpoint             := STRING_TO_INT(GVL_DB.stSysParameters.cal_Replicates);
        GVL_Settings.stCalibParameters.iCalIntervalDays                := STRING_TO_UINT(GVL_DB.stSysParameters.cal_PumpCallIntervalDays);
        GVL_Settings.stCalibParameters.iAirDryTimeSec                  := STRING_TO_UINT(GVL_DB.stSysParameters.AirDryTimeOnCompletation);

        GVL_Settings.bGeneralSealAndPump                               := STRING_TO_BOOL(GVL_DB.stSysParameters.gen_SealAndPump);

        GVL_Settings.stLeakTestParameters.iAllowableLeakTestFailures   := STRING_TO_UINT(GVL_DB.stSysParameters.lkt_AllowableLeakTestFail);
        GVL_Settings.stLeakTestParameters.tLeakTestBuildUpTime         := STRING_TO_UINT(GVL_DB.stSysParameters.lkt_LeakTestBuildupTime);
        GVL_Settings.stLeakTestParameters.tLeakTestMonitorTime         := STRING_TO_UINT(GVL_DB.stSysParameters.lkt_LeakTestHoldTime);
        GVL_Settings.stLeakTestParameters.rLeakTestPressureLimit       := STRING_TO_REAL(GVL_DB.stSysParameters.lkt_LeakTestPressure);

        GVL_Settings.stMachineParam.aM1Position[2]                     := STRING_TO_INT(GVL_DB.stSysParameters.mec_PlatesClosedPosition);
        GVL_Settings.stMachineParam.aM1Position[3]                     := STRING_TO_INT(GVL_DB.stSysParameters.mec_PlatesDryPosition);
        GVL_Settings.stMachineParam.rM1Velocity                        := STRING_TO_LREAL(GVL_DB.stSysParameters.mec_PlatesVelocity);

        GVL_Settings.stPumpParameters.iMeterVelocity                   := STRING_TO_UINT(GVL_DB.stSysParameters.pmp_MeterVelocity);
        GVL_Settings.stPumpParameters.iRunVelocity                     := STRING_TO_UINT(GVL_DB.stSysParameters.pmp_RunVelocity);
        GVL_Settings.stPumpParameters.iEmptyFactor                     := STRING_TO_UINT(GVL_DB.stSysParameters.pmp_EmptyFactor);
        GVL_Settings.stPumpParameters.iFillolventTubesFactor           := STRING_TO_UINT(GVL_DB.stSysParameters.pmp_FillSolventTubesFactor);

        GVL_Settings.stMachineParam.aM3Position[4]                     := STRING_TO_INT(GVL_DB.stSysParameters.smp_AboveCalibration);
        GVL_Settings.stMachineParam.aM3Position[2]                     := STRING_TO_INT(GVL_DB.stSysParameters.smp_AboveVialSet1);
        GVL_Settings.stMachineParam.aM3Position[3]                     := STRING_TO_INT(GVL_DB.stSysParameters.smp_VialSetSpacing);

        GVL_Settings.stMachineParam.aM2Position[4]                     := STRING_TO_INT(GVL_DB.stSysParameters.smp_IntoResBottom);
        GVL_Settings.stMachineParam.aM2Position[5]                     := STRING_TO_INT(GVL_DB.stSysParameters.smp_IntoResDispense);
        GVL_Settings.stMachineParam.aM2Position[6]                     := STRING_TO_INT(GVL_DB.stSysParameters.smp_IntoResWeigh);
        GVL_Settings.stMachineParam.aM2Position[3]                     := STRING_TO_INT(GVL_DB.stSysParameters.smp_IntoVials);
        GVL_Settings.stMachineParam.aM2Position[2]                     := STRING_TO_INT(GVL_DB.stSysParameters.smp_IntoWaste);

        GVL_Settings.bDisplayManualControl                             := STRING_TO_BOOL(GVL_DB.stSysParameters.sec_DisplayManualControl);
        GVL_Settings.bCheckLogonEachRun                                := STRING_TO_BOOL(GVL_DB.stSysParameters.sec_CheckLogonEachRun);

        state := 30;


    30: // REQUEST_LAST_CALIBRATION_ID
    bBusy := TRUE;

		IF NOT bQueryStarted THEN
			DB_Query.state := E_DB_QUERY_STATE.SELECT_LAST_CALIBRATION_ID;
			bQueryStarted := TRUE;
			bDbBusySeen := FALSE;
			tonTimeout(IN := TRUE, PT := tTimeout);
		END_IF
	
		tonTimeout(IN := TRUE, PT := tTimeout);
	
		IF DB_Query.FB_SelectArray.bBusy THEN
			bDbBusySeen := TRUE;
		END_IF
	
		IF bDbBusySeen AND NOT DB_Query.FB_SelectArray.bBusy THEN
			tonTimeout(IN := FALSE);
			bQueryStarted := FALSE;
			bDbBusySeen := FALSE;
			state := 40;
	
		ELSIF tonTimeout.Q THEN
			tonTimeout(IN := FALSE);
			bQueryStarted := FALSE;
			bDbBusySeen := FALSE;
			state := 900;
			nErrorId := 1002;
		END_IF


    40: // REQUEST_LINEAR_MOTORS
		bBusy := TRUE;
	
		IF NOT bQueryStarted THEN
			DB_Query.state := E_DB_QUERY_STATE.SELECT_LINEAR_MOTORS;
			bQueryStarted := TRUE;
			bDbBusySeen := FALSE;
			tonTimeout(IN := TRUE, PT := tTimeout);
		END_IF
	
		tonTimeout(IN := TRUE, PT := tTimeout);
	
		IF DB_Query.FB_SelectArray.bBusy THEN
			bDbBusySeen := TRUE;
		END_IF
	
		IF bDbBusySeen AND NOT DB_Query.FB_SelectArray.bBusy THEN
			tonTimeout(IN := FALSE);
			bQueryStarted := FALSE;
			bDbBusySeen := FALSE;
			state := 50;
	
		ELSIF tonTimeout.Q THEN
			tonTimeout(IN := FALSE);
			bQueryStarted := FALSE;
			bDbBusySeen := FALSE;
			state := 900;
			nErrorId := 1003;
		END_IF


    50: // APPLY_LINEAR_MOTORS
        GVL_HMI.aCalibLinearPumps[1].rNewPosition  := STRING_TO_LREAL(GVL_DB.stLinearMotors.pump1);
        GVL_HMI.aCalibLinearPumps[2].rNewPosition  := STRING_TO_LREAL(GVL_DB.stLinearMotors.pump2);
        GVL_HMI.aCalibLinearPumps[3].rNewPosition  := STRING_TO_LREAL(GVL_DB.stLinearMotors.pump3);
        GVL_HMI.aCalibLinearPumps[4].rNewPosition  := STRING_TO_LREAL(GVL_DB.stLinearMotors.pump4);
        GVL_HMI.aCalibLinearPumps[5].rNewPosition  := STRING_TO_LREAL(GVL_DB.stLinearMotors.pump5);
        GVL_HMI.aCalibLinearPumps[6].rNewPosition  := STRING_TO_LREAL(GVL_DB.stLinearMotors.pump6);
        GVL_HMI.aCalibLinearPumps[7].rNewPosition  := STRING_TO_LREAL(GVL_DB.stLinearMotors.pump7);
        GVL_HMI.aCalibLinearPumps[8].rNewPosition  := STRING_TO_LREAL(GVL_DB.stLinearMotors.pump8);
        GVL_HMI.aCalibLinearPumps[9].rNewPosition  := STRING_TO_LREAL(GVL_DB.stLinearMotors.pump9);
        GVL_HMI.aCalibLinearPumps[10].rNewPosition := STRING_TO_LREAL(GVL_DB.stLinearMotors.pump10);

        GVL_HMI.aCalibLinearPumps[1].rOldPosition  := GVL_Retain.rLinearPumpOldPosition[1];
        GVL_HMI.aCalibLinearPumps[2].rOldPosition  := GVL_Retain.rLinearPumpOldPosition[2];
        GVL_HMI.aCalibLinearPumps[3].rOldPosition  := GVL_Retain.rLinearPumpOldPosition[3];
        GVL_HMI.aCalibLinearPumps[4].rOldPosition  := GVL_Retain.rLinearPumpOldPosition[4];
        GVL_HMI.aCalibLinearPumps[5].rOldPosition  := GVL_Retain.rLinearPumpOldPosition[5];
        GVL_HMI.aCalibLinearPumps[6].rOldPosition  := GVL_Retain.rLinearPumpOldPosition[6];
        GVL_HMI.aCalibLinearPumps[7].rOldPosition  := GVL_Retain.rLinearPumpOldPosition[7];
        GVL_HMI.aCalibLinearPumps[8].rOldPosition  := GVL_Retain.rLinearPumpOldPosition[8];
        GVL_HMI.aCalibLinearPumps[9].rOldPosition  := GVL_Retain.rLinearPumpOldPosition[9];
        GVL_HMI.aCalibLinearPumps[10].rOldPosition := GVL_Retain.rLinearPumpOldPosition[10];

        state := 60;


    60: // REQUEST_LAST_SOLVENT
		bBusy := TRUE;
	
		IF NOT bQueryStarted THEN
			DB_Query.state := E_DB_QUERY_STATE.SELECT_LAST_SOLVENT;
			bQueryStarted := TRUE;
			bDbBusySeen := FALSE;
			tonTimeout(IN := TRUE, PT := tTimeout);
		END_IF
	
		tonTimeout(IN := TRUE, PT := tTimeout);
	
		IF DB_Query.FB_SelectArray.bBusy THEN
			bDbBusySeen := TRUE;
		END_IF
	
		IF bDbBusySeen AND NOT DB_Query.FB_SelectArray.bBusy THEN
			tonTimeout(IN := FALSE);
			bQueryStarted := FALSE;
			bDbBusySeen := FALSE;
			state := 70;
	
		ELSIF tonTimeout.Q THEN
			tonTimeout(IN := FALSE);
			bQueryStarted := FALSE;
			bDbBusySeen := FALSE;
			state := 900;
			nErrorId := 1004;
		END_IF


    70: // APPLY_SOLVENTS
        GVL_HMI.stHMISolventsInfo[1].sSolventName := GVL_DB.stSolvents.solventName1;
        GVL_HMI.stHMISolventsInfo[2].sSolventName := GVL_DB.stSolvents.solventName2;
        GVL_HMI.stHMISolventsInfo[3].sSolventName := GVL_DB.stSolvents.solventName3;
        GVL_HMI.stHMISolventsInfo[4].sSolventName := GVL_DB.stSolvents.solventName4;

        GVL_HMI.stHMISolventsInfo[1].rDensity     := STRING_TO_LREAL(GVL_DB.stSolvents.density1);
        GVL_HMI.stHMISolventsInfo[2].rDensity     := STRING_TO_LREAL(GVL_DB.stSolvents.density2);
        GVL_HMI.stHMISolventsInfo[3].rDensity     := STRING_TO_LREAL(GVL_DB.stSolvents.density3);
        GVL_HMI.stHMISolventsInfo[4].rDensity     := STRING_TO_LREAL(GVL_DB.stSolvents.density4);

        GVL_Settings.stSolventsInfo := GVL_HMI.stHMISolventsInfo;

        state := 100;


    100: // DONE
        bBusy := FALSE;
        bDone := TRUE;
        bError := FALSE;
        tonTimeout(IN := FALSE);

        IF NOT bExecute THEN
            state := 0;
        END_IF


    900: // ERROR
        bBusy := FALSE;
        bDone := FALSE;
        bError := TRUE;
        tonTimeout(IN := FALSE);

        IF bReset THEN
            state := 0;
            bError := FALSE;
            nErrorId := 0;
        END_IF


ELSE
    state := 900;
    nErrorId := 9999;

END_CASE

END_PROGRAM

// ---- POUs/Utilities/PRG_ValveTest.TcPOU
PROGRAM PRG_ValveTest
VAR
	eStep           : INT := 0;
    tWait           : TON;      // Timer de 500 ms
    iCycleCounter   : INT := 0; // Contador de ciclos globais (todas as válvulas)
    iCycleThreshold : INT := 600;

    i               : INT;      // Índice de loop
    bAllDone        : BOOL;     // Flag: todas as válvulas terminaram
END_VAR

// ----- Máquina de Estados -----
CASE eStep OF

    // -------------------------------------------------
    // 0) Mover TODAS as válvulas para posição 1
    // -------------------------------------------------
    0:
        bAllDone := TRUE;

        FOR i := 1 TO 5 DO
            // Se alguma ainda não terminou o movimento, AllDone fica FALSE
            IF NOT GVL_Motion.aValvesObj[i].MoveValve(
                    iPosition := 1,
                    rVelocity := GVL_Motion.aValves[i].rTargetVel,
                    rAcc      := GVL_Motion.aValves[i].rAcceleration,
                    rDec      := GVL_Motion.aValves[i].rDeceleration)
            THEN
                bAllDone := FALSE;
            END_IF
        END_FOR
		

        // Só avança quando TODAS retornarem TRUE
        IF bAllDone THEN
            tWait(IN := FALSE);    // reset do TON
            eStep := 10;
        END_IF

    // -------------------------------------------------
    // 10) Espera 500 ms após TODAS chegarem na posição 1
    // -------------------------------------------------
    10:
        tWait(IN := TRUE, PT := T#500MS);
        IF tWait.Q THEN
            tWait(IN := FALSE);
            eStep := 20;
        END_IF

    // -------------------------------------------------
    // 20) Mover TODAS as válvulas para posição 6
    // -------------------------------------------------
    20:
        bAllDone := TRUE;

        FOR i := 1 TO 5 DO
            IF NOT GVL_Motion.aValvesObj[i].MoveValve(
                    iPosition := 6,
                    rVelocity := GVL_Motion.aValves[i].rTargetVel,
                    rAcc      := GVL_Motion.aValves[i].rAcceleration,
                    rDec      := GVL_Motion.aValves[i].rDeceleration)
            THEN
                bAllDone := FALSE;
            END_IF
        END_FOR

        IF bAllDone THEN
            tWait(IN := FALSE);
            eStep := 30;
        END_IF

    // -------------------------------------------------
    // 30) Espera 500 ms após TODAS chegarem na posição 6
    //      Depois conta 1 ciclo global (todas as 5 passaram por 1→6)
    // -------------------------------------------------
    30:
        tWait(IN := TRUE, PT := T#500MS);
        IF tWait.Q THEN
            tWait(IN := FALSE);

            iCycleCounter := iCycleCounter + 1;

            IF iCycleCounter < iCycleThreshold THEN
                eStep := 0;      // novo ciclo 1→6
            ELSE
                eStep := 100;    // fim dos testes
            END_IF
        END_IF

    // -------------------------------------------------
    // 100) Fim do teste
    // -------------------------------------------------
    100:
        // Aqui você pode colocar:
        // GVL_HMI.bValveTestDone := TRUE; ou algo assim
END_CASE

END_PROGRAM

// ---- POUs/0. Main/MAIN_Events.TcPOU
PROGRAM MAIN_Events
VAR
END_VAR

END_PROGRAM

// ---- POUs/0. Main/MAIN_HMI.TcPOU
PROGRAM MAIN_HMI
VAR
END_VAR

END_PROGRAM

// ---- POUs/0. Main/MAIN_Services.TcPOU
PROGRAM MAIN_Services
VAR
END_VAR

END_PROGRAM

// ---- POUs/5. Calibration/FB_ScaleDevice.TcPOU
FUNCTION_BLOCK FB_ScaleDevice
VAR_INPUT
    sRemoteHost 	: STRING := '192.168.1.100';
    nRemotePort 	: UINT 	 := 8001;
	bExecuteRequest : BOOL;
	rLastWeight     : LREAL;
END_VAR

VAR_OUTPUT
	bWeightReady : BOOL;
    bBusy        : BOOL;
    bError       : BOOL;
    nErrorID     : UDINT;
END_VAR

VAR
    fbTcpClient     : FB_TcpClient;
   
    bRequestDone    : BOOL;
    sRawResponse    : STRING(255);
    
    sLastMessage    : STRING(255);
END_VAR

// Continous call to keep the function block ready for communication 
IF bExecuteRequest OR fbTcpClient.bBusy THEN
	fbTcpClient(
		sRemoteHost := sRemoteHost,
		nRemotePort := nRemotePort,
		bExecute := bExecuteRequest,
		tStateDelay := T#500MS,
		bConnectionDone => bRequestDone,
		sResponse => sRawResponse,
		bError => bError,
		nErrorID => nErrorID
	);
END_IF

// Done and Reset flags
IF fbTcpClient.bConnectionDone THEN
    bExecuteRequest := FALSE;
    rLastWeight := F_ParseWeight(sRawResponse);
    sLastMessage := CONCAT('Weight: ', LREAL_TO_STRING(rLastWeight));
	bWeightReady := TRUE;
END_IF

METHOD RequestWeight : LREAL
VAR_OUTPUT
    bSuccess : BOOL;
    sMessage : STRING;
END_VAR
// Triggering fbTcpClient
IF NOT bExecuteRequest AND NOT fbTcpClient.bBusy THEN
    bExecuteRequest := TRUE;
END_IF
// Releasing fbTcpClient 
IF fbTcpClient.bConnectionDone THEN
    RequestWeight := rLastWeight;
    bSuccess := TRUE;
    sMessage := sLastMessage;
ELSE
    bSuccess := FALSE;
END_IF
END_METHOD

METHOD Reset : BOOL
VAR_INPUT
END_VAR
bWeightReady := FALSE;
bBusy        := FALSE;
bError       := FALSE;
nErrorID     := 0;
bExecuteRequest := FALSE;
bRequestDone    := FALSE;
sRawResponse    := '';
rLastWeight     := 0.0;
sLastMessage    := '';

IF fbTcpClient.Reset() AND NOT bWeightReady THEN
	Reset := TRUE;
ELSE
	Reset := FALSE;
END_IF
END_METHOD

END_FUNCTION_BLOCK

// ---- POUs/Utilities/FB_TCPClient.TcPOU
FUNCTION_BLOCK FB_TCPClient
// This function block handles TCP communication with a scale using MT-SICS commands (e.g., SI) to retrieve weight data.

VAR_INPUT
    sRemoteHost  : T_IPv4Addr;   // IP address of the scale
    nRemotePort  : UINT;         // TCP port of the scale
    bExecute     : BOOL;         // Manual trigger to start communication
    tStateDelay  : TIME := T#100MS; // Delay between state transitions
	sCommand 	 : STRING(16);
END_VAR

VAR_OUTPUT
    bConnected       : BOOL;         // True if connection to scale was established
    sReceivedData_At : STRING(255);  // Raw response received from the scale
	sReceivedData_SI : STRING(255);  // Raw response received from the scale
    sResponse  		 : STRING(255);  // Human-readable description of the response
    fWeight          : REAL;         // Parsed weight value from the scale
    bConnectionDone  : BOOL;         // True when communication finishes successfully or with error
    nErrorID         : UDINT;        // Error ID from socket function blocks
    bError           : BOOL;         // General error flag
    bBusy            : BOOL;         // Indicates communication in progress
    bOperatorCheck   : BOOL;         // True if manual intervention is needed (e.g., scale not ready)
END_VAR

VAR
    iState                  : INT;             // State machine control variable
    fbSocketConnect         : FB_SocketConnect; // Function block to establish TCP connection
    fbSocketSend            : FB_SocketSend;    // Function block to send data over TCP
    fbSocketClose           : FB_SocketClose;   // Function block to close TCP connection
    fbSocketCloseAll        : FB_SocketCloseAll;// Function block to close all TCP connections
    fbSocketReceive_AtCmd   : FB_SocketReceive; // Function block to receive data over TCP
    fbSocketReceive_SI      : FB_SocketReceive;
	fbSocketReceive_SI2		: FB_SocketReceive;
    hSocket                 : T_HSOCKET;        // Socket handle for TCP session

    sSendData               : STRING(10);       // Message to be sent to the scale
    nRecBytes_At            : UDINT;            // Number of bytes received
	nRecBytes_SI			: UDINT; 
    sCRLF                   : STRING(2);        // Carriage return + line feed sequence
    bTriggerPrev            : BOOL;             // Previous state of trigger input
	sReceivedData2			: STRING(255);

    tonStateTimer            : TON;              // Timer for controlling state delays
    tonCloseConnectionTimer: TON;              // Timer for socket close delay
    tonOpenConnectionTimer : TON;              // Timer for socket open delay
    tonSendCommandTimer    : TON;              // Timer for command send delay
    tonReceivingTimer      : TON;              // Timer for response receiving delay
    tonSocketCloseTimer    : TON;              // Timer for socket close finalization

    bCloseConnectionTimer  : BOOL := FALSE;     // Pulse control for close timer
    bOpenConnectionTimer   : BOOL := FALSE;     // Pulse control for open timer
    bSendCommandTimer      : BOOL := FALSE;     // Pulse control for send timer
    bReceivingTimer        : BOOL := FALSE;     // Pulse control for receive timer
    bCloseSocketTimer      : BOOL := FALSE;     // Pulse control for socket close timer
	bResetDone			   : BOOL := FALSE;		// Internal FB Reset Flag
	bTimerOutput		   : BOOL := FALSE;
	bStart				   : BOOL := FALSE;
	bReceiveActive		   : BOOL := FALSE;
	bReceiveExecute		   : BOOL := FALSE;

    tStepTimer              : TIME := T#500ms;  // Default step delay for timers

    receiveTimeout          : INT := 0;         // Timeout counter for receiving response
    MAX_TIMEOUT             : INT := 50;        // Max retries for receive timeout
    retryCount              : INT := 0;         // Number of retry attempts
    MAX_RETRIES             : INT := 2;         // Maximum retry attempts for S I error

    iStart                  : INT := 4;         // Index of first numeric character in response
    iEnd                    : INT := 5;         // Index of end of numeric string
    sWeightStr              : STRING(10);       // Substring extracted for weight conversion
	iSubStep				: UINT;

    fbConnectTrigger        : R_TRIG;           // Rising edge trigger for connect
    fbSendTrigger           : R_TRIG;           // Rising edge trigger for send
    fbReceiveTrigger        : R_TRIG;           // Rising edge trigger for receive
    fbCloseTrigger          : R_TRIG;           // Rising edge trigger for close
    fbCloseAllTrigger       : R_TRIG;           // Rising edge trigger for close all
END_VAR

// --- TCP Client States for Weighing Scale Communication ---

IF NOT bStart AND bExecute THEN
    iState := 0;
    bStart := bExecute;
END_IF

CASE iState OF

    // --- STATE 0: Initial Reset ---
    0:
        IF bStart AND NOT bResetDone THEN
            bResetDone := Reset();
        END_IF

        IF bResetDone THEN
            tonStateTimer(IN := TRUE, PT := tStateDelay);
            IF tonStateTimer.Q THEN
                tonStateTimer(IN := FALSE);
                iState := 5;
                bBusy := TRUE;
            END_IF
        END_IF

    // --- STATE 5: Close All Sockets ---
    5:
        bResetDone := FALSE;
        fbSocketCloseAll(
            sSrvNetId := '',
            bExecute := TRUE,
            tTimeout := T#10S,
            bBusy => bBusy,
            bError => bError,
            nErrId => nErrorID
        );

        tonStateTimer(IN := TRUE, PT := T#1S);
        IF NOT bBusy AND tonStateTimer.Q THEN
            tonStateTimer(IN := FALSE);
            iState := 10;
        END_IF

    // --- STATE 10: TCP Connect ---
    10:
        fbSocketConnect(
            sRemoteHost := sRemoteHost,
            nRemotePort := nRemotePort,
            bExecute := TRUE,
            tTimeout := T#10S,
            bBusy => bBusy,
            bError => bError,
            nErrId => nErrorID,
            hSocket => hSocket
        );

        tonStateTimer(IN := TRUE, PT := T#1S);
        IF NOT fbSocketConnect.bBusy AND tonStateTimer.Q THEN
            IF bError THEN
                sResponse := CONCAT('Connection error! Code: ', UDINT_TO_STRING(nErrorID));
				GVL_Alarms.bTCPCLientConnectError := TRUE;
                iState := 60;
            ELSIF hSocket.handle <> 0 THEN
                bConnected := TRUE;
                iState := 20;
            ELSE
                sResponse := 'No socket handle.';
                iState := 60;
            END_IF
			tonStateTimer(IN := FALSE);
        END_IF

    // --- STATE 20: Send "@" Command ---
    20:
        sSendData := CONCAT('@', CONCAT(CHR(13), CHR(10)));
        fbSocketSend(
            hSocket := hSocket,
            cbLen := SIZEOF(sSendData),
            pSrc := ADR(sSendData),
            bExecute := TRUE,
            tTimeout := T#1S,
            bError => bError,
            nErrId => nErrorID
        );

        tonStateTimer(IN := TRUE, PT := T#1S);
        IF NOT bBusy AND tonStateTimer.Q THEN
            tonStateTimer(IN := FALSE);
			fbSocketSend(bExecute := FALSE);
            iState := 30;
        END_IF
		
		IF fbSocketSend.bError THEN
			sResponse := CONCAT('TCP Socket Send error! Code: ', UDINT_TO_STRING(fbSocketSend.nErrId));
			GVL_Alarms.bTCPCLientSendError := TRUE;
			iState := 60;
		END_IF

    // --- STATE 30: Receive "@" Response ---
    30:
        fbSocketReceive_AtCmd(
            hSocket := hSocket,
            cbLen := SIZEOF(sReceivedData_At),
            pDest := ADR(sReceivedData_At),
            bExecute := TRUE,
            tTimeout := T#3S,
            bError => bError,
            nErrId => nErrorID,
            nRecBytes => nRecBytes_At
        );
		tonStateTimer(IN := TRUE, PT := T#1S);
        IF NOT fbSocketReceive_AtCmd.bBusy AND tonStateTimer.Q THEN
			IF nRecBytes_At > 0 THEN
				fbSocketReceive_AtCmd(bExecute := FALSE);
				iState := 40;
			ELSE
                sResponse := '@_Error';
                iState := 60;
			END_IF
			tonStateTimer(IN := FALSE);
        END_IF
		
		IF fbSocketReceive_AtCmd.bError THEN
			sResponse := CONCAT('TCP Socket Receive error! Code: ', UDINT_TO_STRING(fbSocketReceive_AtCmd.nErrId));
			GVL_Alarms.bTCPCLientReceiveError := TRUE;
			iState := 60;
		END_IF

    // --- STATE 40: Send "SI" Command ---
    40:
        sSendData := CONCAT('SI', CONCAT(CHR(13), CHR(10)));
        fbSocketSend(
            hSocket := hSocket,
            cbLen := SIZEOF(sSendData),
            pSrc := ADR(sSendData),
            bExecute := TRUE,
            tTimeout := T#1S,
            bError => bError,
            nErrId => nErrorID
        );

        tonStateTimer(IN := TRUE, PT := T#1S);
        IF NOT bBusy AND tonStateTimer.Q THEN
            tonStateTimer(IN := FALSE);
            iState := 50;
        END_IF
		
		IF fbSocketSend.bError THEN
			sResponse := CONCAT('TCP Socket Send error! Code: ', UDINT_TO_STRING(fbSocketSend.nErrId));
			GVL_Alarms.bTCPCLientSendError := TRUE;
			iState := 60;
		END_IF

    // --- STATE 50: Receive SI Response ---
    50:
        fbSocketReceive_SI(
            hSocket := hSocket,
            cbLen := SIZEOF(sReceivedData_SI),
            pDest := ADR(sReceivedData_SI),
            bExecute := TRUE,
            tTimeout := T#5S,
            bError => bError,
            nErrId => nErrorID,
            nRecBytes => nRecBytes_SI
        );
		tonStateTimer(IN := TRUE, PT := T#1S);
        IF NOT fbSocketReceive_SI.bBusy AND tonStateTimer.Q THEN
            IF nRecBytes_SI > 0 THEN
                sResponse := sReceivedData_SI;
                iState := 60;
            ELSE
                sResponse := 'SI_Error';
                iState := 60;
            END_IF
			tonStateTimer(in := FALSE);
        END_IF
		
		IF fbSocketReceive_SI.bError THEN
			sResponse := CONCAT('TCP Socket Receive error! Code: ', UDINT_TO_STRING(fbSocketReceive_SI.nErrId));
			GVL_Alarms.bTCPCLientReceiveError := TRUE;
			iState := 60;
		END_IF

    // --- STATE 60: Close socket and finish ---
    60:
        fbSocketClose(
            hSocket := hSocket,
            bExecute := TRUE,
            tTimeout := T#2S,
            bError => bError,
            nErrId => nErrorID
        );

        tonStateTimer(IN := TRUE, PT := T#1S);
        IF NOT bBusy AND tonStateTimer.Q THEN
            tonStateTimer(IN := FALSE);
            bConnectionDone := TRUE;
            bStart := FALSE;
            iState := 0;
        END_IF
		
		IF fbSocketClose.bError THEN
			sResponse := CONCAT('TCP Socket Receive error! Code: ', UDINT_TO_STRING(fbSocketClose.nErrId));
			GVL_Alarms.bTCPCLientCloseError := TRUE;
			iState := 60;
		END_IF

END_CASE

METHOD Reset : BOOL
VAR_INPUT
END_VAR
// Reset method to initialize all function blocks, outputs and timers to default state.
fbSocketConnect(bExecute := FALSE);
fbSocketSend(bExecute := FALSE);
fbSocketReceive_AtCmd(bExecute := FALSE);
fbSocketReceive_SI(bExecute := FALSE);
fbSocketClose(bExecute := FALSE);
fbSocketCloseAll(bExecute := FALSE);

tonStateTimer(IN := FALSE);
TonCloseConnectionTimer(IN := FALSE);
TonOpenConnectionTimer(IN := FALSE);
TonSendCommandTimer(IN := FALSE);
TonReceivingTimer(IN := FALSE);
TonSocketCloseTimer(IN := FALSE);

fbConnectTrigger(CLK := FALSE);
fbSendTrigger(CLK := FALSE);
fbReceiveTrigger(CLK := FALSE);
fbCloseTrigger(CLK := FALSE);
fbCloseAllTrigger(CLK := FALSE);

bCloseConnectionTimer := FALSE;
bOpenConnectionTimer := FALSE;
bSendCommandTimer := FALSE;
bReceivingTimer := FALSE;
bCloseSocketTimer := FALSE;
bTriggerPrev := FALSE;

bTimerOutput := FALSE;
bConnected := FALSE;
bConnectionDone := FALSE;
bBusy := FALSE;
bError := FALSE;
bOperatorCheck := FALSE;
nErrorID := 0;
retryCount := 0;
fWeight := 0;
sResponse := '';
sWeightStr := '';
iStart := 4;
iEnd := 5;

IF NOT fbSocketConnect.bBusy AND NOT fbSocketSend.bBusy AND NOT fbSocketReceive_AtCmd.bBusy AND NOT fbSocketReceive_SI.bBusy AND NOT fbSocketClose.bBusy AND NOT fbSocketCloseAll.bBusy THEN
	Reset := TRUE;
	RETURN;
ELSE
	Reset := FALSE;
END_IF
END_METHOD

END_FUNCTION_BLOCK

// ---- POUs/Functions/F_ParseWeight.TcPOU
FUNCTION F_ParseWeight : LREAL
VAR_INPUT
    sResponse : STRING(255);
END_VAR

VAR
    sCleaned    : STRING(255);
    sValueOnly  : STRING(50);
    iStart      : INT;
    iEnd        : INT;
    i           : INT;
    sChar       : STRING(1);
END_VAR

//Balance's response parse and intepretation
IF LEFT(sResponse, 3) = 'S S' OR LEFT(sResponse, 3) = 'S D' THEN  //Check if the response is a acceptable weigth value
	//Remove controll char of the end of the string (CR LF)
	sResponse := LEFT(sResponse, LEN(sResponse) - 2);
	
	//Look up for the first numeric char (passing initial spaces)
	iStart := 4;  // To begin after the char "S S "
	WHILE (iStart <= LEN(sResponse)) AND MID(sResponse, 1, iStart) = CHR(32) DO
		iStart := iStart + 1;
	END_WHILE;

	//Find ou the number ending (Before weight unit messure)
	iEnd := iStart + 1;
	WHILE (iEnd <= LEN(sResponse)) AND 
	((MID(sResponse, 1, iEnd) <> 'k' OR MID(sResponse, 1, iEnd) <> 'g')) DO
		iEnd := iEnd + 1;
	END_WHILE

	//Back 1 char to not include the weight unit
	iEnd := iEnd - 1;

	//Extract and weigth convertion
	IF (iStart > 0) AND (iEnd >= iStart) THEN
		sValueOnly := MID(sResponse, iEnd - iStart + 1, iStart);  //Extract the wegth without the meassure unit
		F_ParseWeight := STRING_TO_REAL(sValueOnly);  //String to Real convertion
	ELSE
		F_ParseWeight := 9998.0;
	END_IF
ELSE
	F_ParseWeight := 9999.0;
END_IF

END_FUNCTION

// ---- POUs/2. AutoCycle/Hardware Control/FB_SetSolenoid.TcPOU
FUNCTION_BLOCK FB_SetSolenoid
VAR_INPUT
END_VAR
VAR_OUTPUT
END_VAR
VAR
END_VAR

METHOD AirDry : BOOL
VAR_INPUT
END_VAR
AirDry:= FALSE;

GVL_IO.gDigOutputs.bSolenoidValveA := FALSE;
GVL_IO.gDigOutputs.bSolenoidValveB := FALSE;
GVL_IO.gDigOutputs.bSolenoidValveC := TRUE;

GVL_Calibration.eLeakTestState := E_LeakTestState.IDLE;

AirDry := TRUE;
RETURN;
END_METHOD

METHOD HoldPressure : BOOL
VAR_INPUT
END_VAR
HoldPressure:= FALSE;

GVL_IO.gDigOutputs.bSolenoidValveA := TRUE;
GVL_IO.gDigOutputs.bSolenoidValveB := FALSE;
GVL_IO.gDigOutputs.bSolenoidValveC := FALSE;

GVL_Calibration.eLeakTestState := E_LeakTestState.HOLD_PRESSURE;

HoldPressure := TRUE;
RETURN;
END_METHOD

METHOD Idle : BOOL
VAR_INPUT
END_VAR
Idle:= FALSE;

GVL_IO.gDigOutputs.bSolenoidValveA := FALSE;
GVL_IO.gDigOutputs.bSolenoidValveB := FALSE;
GVL_IO.gDigOutputs.bSolenoidValveC := FALSE;

GVL_Calibration.eLeakTestState := E_LeakTestState.IDLE;

Idle := TRUE;
RETURN;
END_METHOD

METHOD PressureUp : BOOL
VAR_INPUT
END_VAR
PressureUp:= FALSE;

GVL_IO.gDigOutputs.bSolenoidValveA := TRUE;
GVL_IO.gDigOutputs.bSolenoidValveB := TRUE;
GVL_IO.gDigOutputs.bSolenoidValveC := FALSE;

GVL_Calibration.eLeakTestState := E_LeakTestState.PRESSURE_UP;

PressureUp := TRUE;
RETURN;
END_METHOD

END_FUNCTION_BLOCK

// ---- POUs/MotionControl/FB_MotorWrapper.TcPOU
FUNCTION_BLOCK FB_MotorWrapper IMPLEMENTS IF_Actuator
VAR_INPUT
END_VAR
VAR_OUTPUT
END_VAR
VAR_IN_OUT
	Axis : AXIS_REF;
END_VAR

VAR
	// MC2 Motion Function Blocks
    fbPower       : MC_Power;
    fbReset       : MC_Reset;
	fbReadStatus  : MC_ReadStatus;
    fbMoveAbs     : MC_MoveAbsolute;
    fbMoveRel     : MC_MoveRelative;
	fbMoveVel	  : MC_MoveVelocity;
	fbSetPos	  : MC_SetPosition;
    fbHome        : MC_Home;
	fbReadPos	  : MC_ReadActualPosition;
    fbStop        : MC_Stop;
	fbHalt		  : MC_Halt;
	fbJog		  : MC_Jog;
    rTrigStop     : R_TRIG;

    fSetPosAbs    : LREAL;
    fSetPosRel    : LREAL;
    bAbsRequest   : BOOL;
    bRelRequest   : BOOL;
    bPowerRequest : BOOL;
    bResetRequest : BOOL;
    bDisableReq   : BOOL;
	
	//Stop()
    bStopExecute     : BOOL;
    bStopRequested   : BOOL;
	bStopDone		 : BOOL;
	
	//GetStatus()
    stStatus       	 : ST_ActuatorStatus;
	stReadStatus	 : ST_AxisReadStatus;
	lastPosition 	 : LREAL := 0.0;
	deltaPos 		 : LREAL;
    bDetectedMovement: BOOL  := FALSE;
    debugSensorValue : BOOL;
	
	//Home()
	bStartDelay		 : BOOL := FALSE;
	tonHoming 		 : TON;
	bhomeExecute	 : BOOL := FALSE;
	bHomeRequest 	 : BOOL := FALSE;

	bExecuteMove	 : BOOL;
	bHomeSensorValue : BOOL;
	bHomeInProgress  : BOOL := FALSE;
	bStartMoveVel	 : BOOL;
	bWaitingForSensorOff : BOOL;
	bWaitingForStop	: BOOL;
	bStartHoming	: BOOL;
	
	//ReadStatus()
	bReadStatusExecute 	: BOOL;
    bReadStatusRequested: BOOL;
	
	//MoveAbs()
	bMoveAbsExecute 	: BOOL;
    bMoveAbsRequested 	: BOOL;
	bMoveAbsDone		: BOOL;
	bMoveAbsStarted		: BOOL;
	rtMoveAbsDone 		: R_TRIG; 
    tonMoveAbs    		: TON;    
    tMoveAbsTout  		: TIME := T#60S;
	tonAbsInWin         : TON;         // estabilidade da janela de posição
	rAbsPosTol          : LREAL := 0.001; // tolerância (ajuste ao teu unit)
	tAbsStable          : TIME  := T#100MS; // estabilidade da janela
	tonAbsTimeout       : TON;         // timeout opcional
	tAbsTimeout         : TIME  := T#60S;   // ajuste conforme curso do eixo
	fbReadVel        	: MC_ReadActualVelocity; // se ainda não existir no FB
	tonVelStill      	: TON;                   // estabilidade de "velocidade ~ 0"
	vTolStill        	: LREAL := 0.0001;       // tolerância de velocidade
	rVelAbs          	: LREAL;                 // auxiliar
	rActPrev         	: LREAL;                 // opcional, se preferir medir Δpos
	
	
	//MoveRel()
	bMoveRelExecute 	: BOOL;
    bMoveRelRequested 	: BOOL;
	bMoveRelDone		: BOOL;
	
	//MoveValve()
	rTargetAngle		: LREAL;
	bMoveValveExecute 	: BOOL;
    bMoveValveRequested : BOOL;
	
	//MoveVel()
	bMoveVelExecute 	: BOOL;
    bMoveVelRequested 	: BOOL;
	bMoveVelDone		: BOOL;
	
	//Reset()
	bResetExecute 		: BOOL;
    bResetRequested 	: BOOL;
	bResetDone			: BOOL;
	
	//SetPosition()
	bSetPosExecute 		: BOOL;
    bSetPosRequested	: BOOL;
	bSetPosDone			: BOOL;
	
	
END_VAR

METHOD Disable : BOOL
VAR_INPUT
END_VAR
// Disable (Remove power from axis)
fbPower(Axis := Axis, Enable := FALSE);
stStatus.bEnabled := FALSE;
stStatus.eState := E_ActuatorState.eDisabled;
Disable := TRUE;
END_METHOD

METHOD Enable : BOOL
VAR_INPUT
END_VAR
// Call MC_Power to enable axis
fbPower(Axis := Axis, Enable := TRUE, Enable_Positive := TRUE, Enable_Negative := TRUE);
stStatus.bEnabled := fbPower.Status;
stStatus.bError := fbPower.Error;
stStatus.iErrorCode := fbPower.ErrorID;
IF fbPower.Error THEN
	stStatus.eState := E_ActuatorState.eError;
	stStatus.sMessage := 'Error in PowerUp';
ELSE
	stStatus.eState := E_ActuatorState.eActive;
END_IF;

Enable := fbPower.Status;
END_METHOD

METHOD GetPosition : LREAL
VAR_INPUT
END_VAR
//Get Actual Position of the motor
//fbReadPos(Axis := Axis, Enable := TRUE);
GetPosition := Axis.NcToPlc.ActPos;
END_METHOD

METHOD GetStatus : ST_ActuatorStatus
VAR_INPUT
END_VAR
// Get unified status struct with all feedback for HMI/diagnostics
fbReadPos(Axis := Axis, Enable := TRUE);
stStatus.fPosition := fbReadPos.Position;
stStatus.bBusy := fbMoveAbs.Busy OR fbMoveRel.Busy OR fbHome.Busy OR fbMoveVel.Busy OR bDetectedMovement;
stStatus.bDone := fbMoveAbs.Done OR fbMoveRel.Done OR fbHome.Done;
stStatus.bError := Axis.Status.Error;

// Calc the position diference
deltaPos := fbReadPos.Position - lastPosition;

IF ABS(deltaPos) > 0.1 THEN
    // Detects forward movement
    IF deltaPos > 0 THEN
		stStatus.bMovingFwd := TRUE;
		stStatus.bMovingBck := FALSE;
		bDetectedMovement   := TRUE;
    // Detects backward movement
    ELSIF deltaPos < 0 THEN
        stStatus.bMovingFwd := FALSE;
        stStatus.bMovingBck := TRUE;
		bDetectedMovement   := TRUE;
    END_IF
ELSE
    // No movement
    stStatus.bMovingFwd := FALSE;
    stStatus.bMovingBck := FALSE;
	bDetectedMovement   := FALSE;
END_IF

lastPosition := fbReadPos.Position;

// Prioritize error messages by source
IF stStatus.bError THEN
	stStatus.eState := E_ActuatorState.eError;
	IF fbPower.Error THEN
		stStatus.sMessage := 'Error in PowerUp';
	ELSIF fbMoveAbs.Error THEN
		stStatus.sMessage := 'Error in MoveAbsolute';
	ELSIF fbMoveRel.Error THEN
		stStatus.sMessage := 'Error in MoveRelative';
	ELSIF fbMoveVel.Error THEN
		stStatus.sMessage := 'Error in MoveVelocity';
	ELSIF fbHome.Error THEN
		stStatus.sMessage := 'Error in Home';
	END_IF
END_IF;

//return
GetStatus := stStatus;
END_METHOD

METHOD Home : BOOL
VAR_INPUT
	pHomeSensor : POINTER TO BOOL; // home sensor pointer
	rVelocity : LREAL;
    rAcc      : LREAL;
    rDec      : LREAL;
	
END_VAR
VAR
	 rTrigHome : R_TRIG;
	 rTrigMove : R_TRIG;
	 rTrigStop : R_TRIG;
END_VAR
bHomeSensorValue  := pHomeSensor^;
IF NOT bHomeRequest THEN
	Home := FALSE;
	bHomeRequest := TRUE;
END_IF

//IF NOT GVL_Motion.bInitialHomingDone THEN
	
	IF bHomeRequest AND NOT bHomeInProgress AND bHomeSensorValue THEN
		bExecuteMove 	:= TRUE;
		bHomeInProgress := TRUE;
	END_IF
	
	IF bHomeRequest AND NOT bHomeInProgress THEN
		bExecuteMove 	:= FALSE;
	
		// If the sensor is already active, skip movement and go to homing directly
		IF NOT bHomeSensorValue THEN
			bStartDelay := TRUE;
			bHomeInProgress := TRUE;
		ELSE
			bExecuteMove := TRUE;
			bHomeInProgress := TRUE;
		END_IF
	END_IF
	
	fbMoveVel(Axis := Axis, Execute := bExecuteMove, Velocity := rVelocity, Acceleration := rAcc, Deceleration := rDec, direction := 1); 
	
	fbStop(Axis := Axis, Execute := bStopExecute, Deceleration := 100);
	
	IF bHomeSensorValue THEN
		//fbMoveVel(Axis := Axis, Execute := bExecuteMove, Velocity := rVelocity, Acceleration := rAcc, Deceleration := rDec, direction := 1); //15, 20, 20
		stStatus.sMessage := 'Seeking home sensor...';
		bStopExecute := FALSE;
	ELSIF NOT bStartDelay THEN
		bExecuteMove := FALSE;
		bStopExecute := TRUE;
		//fbStop(Axis := Axis, Execute := bStopExecute, Deceleration := 10);
	END_IF
	
	IF fbStop.Done THEN
		bStopExecute := FALSE;
		bStartDelay := TRUE;
	END_IF
	
	IF NOT fbStop.Busy THEN
		tonHoming(IN := bStartDelay, PT := T#2S);
	END_IF
	
	IF tonHoming.Q THEN
		bhomeExecute := TRUE;
		stStatus.sMessage := 'Executing MC_Home...';
	END_IF
	
	fbHome(Axis := Axis, Execute := bhomeExecute, Position := 0.0, HomingMode := MC_Direct);
	
	IF fbHome.Done THEN
		stStatus.eState := E_ActuatorState.eIdle;
		stStatus.bError := FALSE;
		stStatus.bDone := TRUE;
		stStatus.sMessage := 'Homing completed';
		bStartDelay  := FALSE;
		bhomeExecute := FALSE;
		tonHoming.IN := FALSE;
		bHomeInProgress := FALSE;
		//GVL_Motion.bMotorsHomeDone := TRUE;
		bHomeRequest := FALSE;
		Home := TRUE;
		RETURN;
	ELSIF fbHome.Error THEN
		stStatus.eState := E_ActuatorState.eError;
		stStatus.bError := TRUE;
		stStatus.iErrorCode := fbHome.ErrorID;
		stStatus.sMessage := 'Error in Homing';
		bhomeExecute := FALSE;
		bStartDelay  := FALSE;
		tonHoming.IN := FALSE;
		bHomeInProgress := FALSE;
		bHomeRequest := FALSE;
		Home := FALSE;
	ELSE
		Home := FALSE;
	END_IF
(*ELSE
	
	IF fbMoveAbs.Done THEN 
		bHomeinProgress := FALSE;
		Home := TRUE;
	END_IF
	
	rTrigMove(CLK := bHomeRequest AND NOT bHomeInProgress);
	
	// If homing previously done then Move to zero position
	fbMoveAbs(Axis := Axis, Execute := rTrigMove.Q, Position := 0, velocity := 15, Acceleration := 15, Deceleration := 15);
	bHomeinProgress := TRUE;
	

	
END_IF*)
END_METHOD

METHOD Jog : BOOL
VAR_INPUT
	bFwd : BOOL;
	bBwd : BOOL;
	//rVelocity : LREAL;
END_VAR
// Call the internal motion block
fbJog(
    Axis := Axis,
    JogForward := bFwd,
    JogBackwards := bBwd,
    Mode := MC_JOGMODE_STANDARD_FAST,
);

// Update actuator status
stStatus.bBusy := fbJog.Busy;
stStatus.bDone := fbJog.Done;
stStatus.bError := fbJog.Error;
stStatus.iErrorCode := fbJog.ErrorID;

Jog := fbJog.Busy;
END_METHOD

METHOD MoveAbsolute : BOOL
VAR_INPUT
	rPosition : LREAL;
    rVelocity : LREAL := 10.0;
    rAcc      : LREAL := 20.0;
    rDec      : LREAL := 20.0;
END_VAR
VAR
	rAct : LREAL;
    rErr : LREAL;
    bInWin : BOOL;
    bStandStill : BOOL;
	opts : ST_MoveOptions;
END_VAR
//Standard Output
MoveAbsolute := FALSE;

// Trigger the command request
IF NOT bMoveAbsRequested THEN
    bMoveAbsExecute := TRUE;
    bMoveAbsRequested := TRUE;
END_IF

// MC_MoveAbsolute function block call
opts.IgnorePositionMonitoring := TRUE;   // Standard practice for move commands

fbMoveAbs(
    Axis := Axis,
    Position := rPosition,
    Execute := bMoveAbsExecute, // Execute flag is controlled by the logic below
    Velocity := rVelocity,
    Acceleration := rAcc,
    Deceleration := rDec,
	options := opts
);

// Release the Execute signal once the block gets in busy or error mode
IF fbMoveAbs.Busy OR fbMoveAbs.Error OR fbMoveAbs.CommandAborted THEN
    bMoveAbsExecute := FALSE;
END_IF

// Flag that movement has successfully started
IF fbMoveAbs.Busy THEN
    bMoveAbsStarted := TRUE;
END_IF

// Status mapping to the wrapper's public status structure
stStatus.bBusy := fbMoveAbs.Busy;
stStatus.bDone := fbMoveAbs.Done;
stStatus.bError := fbMoveAbs.Error;
stStatus.iErrorCode := fbMoveAbs.ErrorID;

//Check if there was any erros on the fbMoveAbs block and resets the trigger
IF bMoveAbsRequested AND bMoveAbsStarted AND 
   	NOT fbMoveAbs.Busy AND NOT fbMoveAbs.Done AND NOT fbMoveAbs.Error THEN
		bMoveAbsRequested := FALSE;
    	bMoveAbsStarted := FALSE;
	
		stStatus.bError := TRUE;
		stStatus.iErrorCode := 9001; // Custom code for 'Motion Aborted/Stuck'
		stStatus.sMessage := 'Movement started but was silently aborted (check external Stop/Power).';
END_IF
	
// Finalization — true Done confirmation
IF bMoveAbsRequested AND fbMoveAbs.Done AND bMoveAbsStarted THEN
    bMoveAbsRequested := FALSE;
	bMoveAbsStarted := FALSE;
    MoveAbsolute := TRUE;
    RETURN;
END_IF

// Abort/error handling
IF fbMoveAbs.CommandAborted THEN
    stStatus.eState := E_ActuatorState.eError;
    stStatus.sMessage := 'Command aborted';
END_IF
IF fbMoveAbs.Error THEN
    stStatus.eState := E_ActuatorState.eError;
    stStatus.sMessage := 'Error in Move Motor';
END_IF
END_METHOD

METHOD MoveRelative : BOOL
VAR_INPUT
	Distance : LREAL;
    Velocity : LREAL := 10.0;
    Acc      : LREAL := 20.0;
    Dec      : LREAL := 20.0;
END_VAR
VAR
END_VAR
// Reuse the same logic from MoveAbsolute
IF NOT bMoveRelRequested THEN
    bMoveRelExecute := TRUE;
    bMoveRelRequested := TRUE;
END_IF

IF fbMoveRel.Busy THEN
    bMoveRelExecute := FALSE;
END_IF

// Call the internal motion block
fbMoveRel(
    Axis := Axis,
    Distance := Distance,
    Execute := bMoveRelExecute,
    Velocity := Velocity,
    Acceleration := Acc,
    Deceleration := Dec
);

// Update actuator status
stStatus.bBusy := fbMoveRel.Busy;
stStatus.bDone := fbMoveRel.Done;
stStatus.bError := fbMoveRel.Error;
stStatus.iErrorCode := fbMoveRel.ErrorID;

IF fbMoveRel.Error THEN
    stStatus.eState := E_ActuatorState.eError;
    stStatus.sMessage := 'Error in Move Motor';
END_IF

IF bMoveRelRequested AND NOT fbMoveRel.Busy AND NOT fbMoveRel.Error THEN
    bMoveRelRequested := FALSE;
    MoveRelative := TRUE;
    RETURN;
ELSE
    MoveRelative := FALSE;
END_IF
END_METHOD

METHOD MoveValve : BOOL
VAR_INPUT
	iPosition : USINT;
	rVelocity : LREAL;
	rAcc	  : LREAL;
	rDec	  : LREAL;
END_VAR
// Map logical valve position to angular position
CASE iPosition OF
    1: rTargetAngle := 0.0;
    2: rTargetAngle := 1200.0;
    3: rTargetAngle := 2400.0;
    4: rTargetAngle := 3600.0;
    5: rTargetAngle := 4800.0;
    6: rTargetAngle := 6000.0;
ELSE
    rTargetAngle := 0;
END_CASE

// Reuse the same logic from MoveAbsolute
IF NOT bMoveValveRequested THEN
    bMoveValveExecute := TRUE;
    bMoveValveRequested := TRUE;
END_IF


// Call the internal motion block
fbMoveAbs(
    Axis := Axis,
    Position := rTargetAngle,
    Execute := bMoveValveExecute,
    Velocity := rVelocity,
    Acceleration := rAcc,
    Deceleration := rDec
);

// Update actuator status
stStatus.bBusy := fbMoveAbs.Busy;
stStatus.bDone := fbMoveAbs.Done;
stStatus.bError := fbMoveAbs.Error;
stStatus.iErrorCode := fbMoveAbs.ErrorID;

IF fbMoveAbs.Busy THEN
    bMoveValveExecute := FALSE;
END_IF

IF fbMoveAbs.Error THEN
    stStatus.eState := E_ActuatorState.eError;
    stStatus.sMessage := 'Error in MoveValve';
END_IF

IF bMoveValveRequested AND NOT fbMoveAbs.Busy AND NOT fbMoveAbs.Error THEN
    bMoveValveRequested := FALSE;
    MoveValve := TRUE;
    RETURN;
ELSE
    MoveValve := FALSE;
END_IF
END_METHOD

METHOD MoveVelocity : BOOL
VAR_INPUT
    rVelocity  : LREAL := 10.0;
    rAcc       : LREAL := 20.0;
    rDec       : LREAL := 20.0;
	iDirection : E_PumpDirection;
END_VAR

VAR
	mcDirection: MC_Direction;
END_VAR
// Reuse the same logic from MoveAbsolute
IF NOT bMoveVelRequested THEN
    bMoveVelExecute := TRUE;
    bMoveVelRequested := TRUE;
END_IF

// Get the corect direction
IF iDirection = E_PumpDirection.Forward THEN
	mcDirection := MC_Direction.MC_Positive_Direction;
	ELSE IF iDirection = E_PumpDirection.Backward THEN
		mcDirection := MC_Direction.MC_Negative_Direction;
	ELSE
		mcDirection := MC_Direction.MC_Current_Direction;
	END_IF
END_IF

// Call the internal motion block
fbMoveVel( 	Axis := Axis,
			Execute := bMoveVelExecute,
			Velocity := rVelocity,
			Direction := mcDirection,
			Acceleration := rAcc,
			Deceleration := rDec
);
			
// Update actuator status
stStatus.bBusy := fbMoveVel.Busy;
stStatus.bError := fbMoveVel.Error;
stStatus.iErrorCode := fbMoveVel.ErrorID;

IF fbMoveVel.Busy THEN
    bMoveVelExecute := FALSE;
END_IF

IF fbMoveVel.Error THEN
    stStatus.eState := E_ActuatorState.eError;
    stStatus.sMessage := 'Error in Move Motor';
END_IF

IF bMoveVelRequested AND NOT fbMoveVel.Busy AND NOT fbMoveVel.Error THEN
    bMoveVelRequested := FALSE;
    MoveVelocity := TRUE;
    RETURN;
ELSE
    MoveVelocity := FALSE;
END_IF
END_METHOD

METHOD ReadStatus : ST_AxisReadStatus
VAR_INPUT
END_VAR
//Method to read status by MC_ReadStatus
Axis.ReadStatus();

//Filling up stReadStatus
stReadStatus.Disabled :=  Axis.Status.Disabled;
stReadStatus.Error := Axis.Status.Error;
stReadStatus.ErrorID := Axis.Status.ErrorID;
stReadStatus.Homed := Axis.Status.Homed;
stReadStatus.Operational := Axis.Status.Operational;
stReadStatus.StandStill := Axis.Status.StandStill;

//Return
ReadStatus := stReadStatus;
END_METHOD

METHOD ReadValveStatus : BOOL
VAR
	cAxisPowerErrorID : UDINT := 16#00004466;
END_VAR
// Read Axis status
Axis.ReadStatus();
(*
// False if there is any power source fail or power fault axis error 
ReadValveStatus :=
    NOT GVL_IO.bPowerSupplyDropSignal
    AND NOT Axis.Status.Error
    AND NOT Axis.Status.ErrorStop
    AND NOT Axis.Status.DriveDeviceError;
*)
//ReadValveStatus := (*NOT Axis.Status.Disabled AND*) NOT (Axis.Status.Error AND Axis.Status.ErrorID = cAxisPowerErrorID);

ReadValveStatus := (NOT Axis.Status.Error) AND (NOT Axis.Status.Disabled);
END_METHOD

METHOD Reset : BOOL
VAR_INPUT
END_VAR
VAR
    (* Local helper to clear flags only on very first call of this reset cycle *)
    bFirstCall : BOOL := FALSE;
	stAxisStat : ST_AxisReadStatus;
END_VAR
// ============================================================================
// 0) Default
// ============================================================================
Reset := FALSE;

// Allways read the actual axis state
Axis.ReadStatus();
stAxisStat.Disabled   			:= Axis.Status.Disabled;
stAxisStat.Error      			:= Axis.Status.Error;
stAxisStat.ErrorID    			:= Axis.Status.ErrorID;
stAxisStat.Homed      			:= Axis.Status.Homed;
stAxisStat.Operational			:= Axis.Status.Operational;
stAxisStat.StandStill 			:= Axis.Status.StandStill;
stAxisStat.MotionCommandsLocked	:= Axis.Status.MotionCommandsLocked;

// 0.1) If the axis is NOT in error, there is nothing to reset.
IF NOT stAxisStat.Error AND NOT stAxisStat.MotionCommandsLocked THEN
    // It guarantees a "clean" status.
    stStatus.bError      := FALSE;
    stStatus.iErrorCode  := 0;
    stStatus.sMessage    := '';
    stStatus.eState      := E_ActuatorState.eIdle;

    // Clear internal reset flags
    bResetRequested      := FALSE;
    bResetExecute        := FALSE;
    bResetDone           := FALSE;

    Reset := TRUE;
    RETURN;
END_IF

// ============================================================================
// 1) Detect new Reset() cycle
// 		- Only enters this section when there is actually an error on the axis
// ============================================================================
IF NOT bResetRequested AND NOT bResetExecute AND NOT bResetDone THEN
    bFirstCall     := TRUE;
    bResetRequested:= TRUE;
END_IF

IF bFirstCall THEN
    // --------------------------------------------------------
    // 1.1) Clears all MC's Executes and internal flags.
    // --------------------------------------------------------
    fbPower(Axis := Axis, Enable := FALSE, Enable_Positive := FALSE, Enable_Negative := FALSE);
    fbMoveAbs(Axis := Axis, Execute := FALSE);
    fbMoveRel(Axis := Axis, Execute := FALSE);
    fbMoveVel(Axis := Axis, Execute := FALSE);
    fbHome(Axis := Axis, Execute := FALSE);
    fbSetPos(Axis := Axis, Execute := FALSE);
    fbStop(Axis := Axis, Execute := FALSE);
    fbHalt(Axis := Axis, Execute := FALSE);
    fbReadStatus(Axis := Axis, Enable := FALSE);
    fbReadPos(Axis := Axis, Enable := FALSE);
	fbReset(Axis := Axis, Execute := FALSE);

    bPowerRequest         := FALSE;
    bDisableReq           := FALSE;

    bAbsRequest           := FALSE;
    bRelRequest           := FALSE;

    bReadStatusRequested  := FALSE;
    bReadStatusExecute    := FALSE;

    // Move Abs
    bMoveAbsRequested     := FALSE;
    bMoveAbsExecute       := FALSE;
    bMoveAbsDone          := FALSE;
    bMoveAbsStarted       := FALSE;

    // Move Rel
    bMoveRelRequested     := FALSE;
    bMoveRelExecute       := FALSE;
    bMoveRelDone          := FALSE;

    // Move Valve
    bMoveValveRequested   := FALSE;
    bMoveValveExecute     := FALSE;

    // Move Vel
    bMoveVelRequested     := FALSE;
    bMoveVelExecute       := FALSE;
    bMoveVelDone          := FALSE;

    // SetPos
    bSetPosRequested      := FALSE;
    bSetPosExecute        := FALSE;
    bSetPosDone           := FALSE;

    // Stop / Halt / Home
    bStopRequested        := FALSE;
    bStopExecute          := FALSE;
    bStopDone             := FALSE;
    bHomeRequest          := FALSE;
    bHomeInProgress       := FALSE;
    bStartHoming          := FALSE;
    bStartMoveVel         := FALSE;
    bWaitingForSensorOff  := FALSE;
    bWaitingForStop       := FALSE;

    // Flags do reset
    bResetRequest         := FALSE;
    bResetRequested       := TRUE;
    bResetDone            := FALSE;

    tonMoveAbs(IN := FALSE);
    tonAbsInWin(IN := FALSE);
    tonHoming(IN := FALSE);
    tonVelStill(IN := FALSE);
    tonAbsTimeout(IN := FALSE);

    rtMoveAbsDone(CLK := FALSE);
    rTrigStop(CLK := FALSE);

    stStatus.bBusy        := FALSE;
    stStatus.bError       := TRUE;             // still error
    stStatus.iErrorCode   := stAxisStat.ErrorID;
    stStatus.sMessage     := 'Resetting axis error...';
    stStatus.eState       := E_ActuatorState.eError;

    bFirstCall := FALSE;
END_IF

// ============================================================================
// 2) Triggers MC_Reset 1x per reset cycle
// ============================================================================
IF bResetRequested AND NOT bResetExecute AND NOT bResetDone THEN
    bResetExecute := TRUE;
END_IF

fbReset(
    Axis    := Axis,
    Execute := bResetExecute
);

// ============================================================================
// 3) MC_Reset error handling
// ============================================================================
IF fbReset.Error THEN
    stStatus.bError      := TRUE;
    stStatus.iErrorCode  := fbReset.ErrorID;
    stStatus.sMessage    := 'Error in MC_Reset';
    stStatus.eState      := E_ActuatorState.eError;

    bResetExecute        := FALSE;
    bResetRequested      := FALSE;
    bResetDone           := FALSE;

    Reset := FALSE;
    RETURN;
END_IF

// MC_Reset's Done
IF fbReset.Done THEN
    bResetExecute := FALSE;
    bResetDone    := TRUE;
END_IF

// ============================================================================
// 4) Finalization: only concludes if the axis really recovered from the error.
// ============================================================================
IF bResetDone AND NOT fbReset.Busy THEN
    // reads the axis status again
    Axis.ReadStatus();
    IF NOT Axis.Status.Error THEN
        // Success
        stStatus.bError      := FALSE;
        stStatus.iErrorCode  := 0;
        stStatus.sMessage    := '';
        stStatus.eState      := E_ActuatorState.eIdle;

        bResetRequested      := FALSE;
        bResetDone           := FALSE;

        Reset := TRUE;
        RETURN;
    ELSE
        // Still in error (e.g., 0x4650, 0x4260, etc.)
		// Starts another MC_Reset cycle
        bResetDone     := FALSE;
        bResetExecute  := TRUE;
        // Reset remains FALSE until the error is actually cleared.
    END_IF
END_IF


(* Old Reset procedure before 2025's Nov27th
// ============================================================================
// 0) Default return
// ============================================================================
Reset := FALSE;

// ============================================================================
// 1) First call of Reset() in this cycle: clear ALL internal flags and MC executes
// ============================================================================

// If neither a reset request nor a reset execution is active, this is a NEW reset cycle
IF NOT bResetRequested AND NOT bResetExecute AND NOT bResetDone THEN
    bFirstCall := TRUE;
    bResetRequested := TRUE;
END_IF

IF bFirstCall THEN
    // ------------------------------------------------------------
    // 1.1) Clear all MC function block Execute flags
    // ------------------------------------------------------------
    fbPower(Axis := Axis, Enable := FALSE, Enable_Positive := FALSE, Enable_Positive := FALSE);   // Optionally remove power - adapt to your logic
    fbMoveAbs(Axis := Axis, Execute := FALSE);
    fbMoveRel(Axis := Axis, Execute := FALSE);
    fbMoveVel(Axis := Axis, Execute := FALSE);
    fbHome(Axis := Axis, Execute := FALSE);
    fbSetPos(Axis := Axis, Execute := FALSE);
    fbStop(Axis := Axis, Execute := FALSE);
    fbHalt(Axis := Axis, Execute := FALSE);
    fbReadStatus(Axis := Axis, Enable := FALSE);
    fbReadPos(Axis := Axis, Enable := FALSE);

    // ------------------------------------------------------------
    // 1.2) Clear general request / state flags (adapt / extend as needed)
    // ------------------------------------------------------------
    bPowerRequest         := FALSE;
    bDisableReq           := FALSE;

    bAbsRequest           := FALSE;
    bRelRequest           := FALSE;

    bReadStatusRequested  := FALSE;
    bReadStatusExecute    := FALSE;

    // Move Absolute
    bMoveAbsRequested     := FALSE;
    bMoveAbsExecute       := FALSE;
    bMoveAbsDone          := FALSE;
    bMoveAbsStarted       := FALSE;

    // Move Relative
    bMoveRelRequested     := FALSE;
    bMoveRelExecute       := FALSE;
    bMoveRelDone          := FALSE;

    // Move Valve / indexing moves
    bMoveValveRequested   := FALSE;
    bMoveValveExecute     := FALSE;

    // Move Velocity
    bMoveVelRequested     := FALSE;
    bMoveVelExecute       := FALSE;
    bMoveVelDone          := FALSE;

    // Set Position
    bSetPosRequested      := FALSE;
    bSetPosExecute        := FALSE;
    bSetPosDone           := FALSE;

    // Stop / Halt / Jog
    bStopRequested        := FALSE;
    bStopExecute          := FALSE;
    bStopDone             := FALSE;

    // Home-related flags
    bStartHoming          := FALSE;
    bHomeInProgress       := FALSE;
    bHomeRequest          := FALSE;
    bStartMoveVel         := FALSE;
    bWaitingForSensorOff  := FALSE;
    bWaitingForStop       := FALSE;

    // Reset request flags themselves
    bResetRequest         := FALSE;   // if you use this one
    bResetRequested       := TRUE;    // mark that we are inside a reset cycle
    bResetDone            := FALSE;

    // ------------------------------------------------------------
    // 1.3) Clear timers / edge detectors (only inputs; they reset themselves)
    // ------------------------------------------------------------
    tonMoveAbs(IN := FALSE);
    tonAbsInWin(IN := FALSE);
    tonHoming(IN := FALSE);
    tonVelStill(IN := FALSE);
	tonAbsTimeout(IN := FALSE);       

	rtMoveAbsDone(CLK := FALSE);
    rTrigStop(CLK := FALSE);

    // ------------------------------------------------------------
    // 1.4) Clear public status structure
    // ------------------------------------------------------------
    stStatus.bBusy        := FALSE;
    stStatus.bError       := FALSE;
    stStatus.iErrorCode   := 0;
    stStatus.sMessage     := '';
    stStatus.eState       := E_ActuatorState.eIdle; // Back to idle after a successful reset

    // First call handled
    bFirstCall := FALSE;
END_IF

// ============================================================================
// 2) Trigger MC_Reset once per reset cycle
// ============================================================================

// If we still did not start fbReset in this cycle, raise Execute edge
IF bResetRequested AND NOT bResetExecute AND NOT bResetDone THEN
    bResetExecute := TRUE;
END_IF;

// Call MC_Reset
fbReset(
    Axis    := Axis,
    Execute := bResetExecute
);

// ============================================================================
// 3) Handle fbReset state: Busy / Done / Error
// ============================================================================

// 3.1) Error handling
IF fbReset.Error THEN
    stStatus.bError       := TRUE;
    stStatus.iErrorCode   := fbReset.ErrorID;
    stStatus.sMessage     := 'Error in MC_Reset';
    stStatus.eState       := E_ActuatorState.eError;

    // Cancel reset cycle on error
    bResetExecute         := FALSE;
    bResetRequested       := FALSE;
    bResetDone            := FALSE;

    // Return FALSE (reset failed)
    Reset := FALSE;
    RETURN;
END_IF

// 3.2) Normal completion
IF fbReset.Done THEN
    // Drop Execute after Done
    bResetExecute := FALSE;
    bResetDone    := TRUE;
END_IF

// ============================================================================
// 4) Finalization and single-pulse TRUE on function return
// ============================================================================

// When reset is marked as done and fbReset is no longer busy, close the cycle
IF bResetDone AND NOT fbReset.Busy THEN
    // Clear internal reset state for next time
    bResetRequested   := FALSE;
    bResetDone        := FALSE;

    // Optionally ensure axis is not in error and not moving here (if needed)

    // Return TRUE exactly once to the caller
    Reset := TRUE;
	RETURN;
END_IF
*)

(* Old Reset procedure before 2025's Nov24th
// =================================================================================================
// 1) Clear all MC_* Execute flags
// =================================================================================================
fbMoveAbs.Execute := FALSE;
fbMoveRel.Execute := FALSE;
fbMoveVel.Execute := FALSE;
fbHome.Execute    := FALSE;
fbStop.Execute    := FALSE;

// =================================================================================================
// 2) Clear internal request/control flags
// =================================================================================================
bMoveAbsRequested := FALSE;
bMoveRelRequested := FALSE;
bMoveVelRequested := FALSE;
bHomeRequest      := FALSE;

bMoveAbsExecute := FALSE;
bMoveRelExecute := FALSE;
bMoveVelExecute := FALSE;
bHomeExecute    := FALSE;
bStopExecute    := FALSE;

bStopRequested  := FALSE;
bStopDone       := FALSE;

// =================================================================================================
// 3) Reset exposed status (optional, for clean diagnostics after reset)
// =================================================================================================
stStatus.bBusy      := FALSE;
stStatus.bError     := FALSE;
stStatus.iErrorCode := 0;
stStatus.sMessage   := '';
// stStatus.eState  := E_ActuatorState.eIdle;  // keep or set later when success

// =================================================================================================
// 4) Build a clean one-scan pulse for MC_Reset via parameter call
// =================================================================================================

// Generates the pulse just once when it's called
IF NOT bResetRequested THEN
    bResetExecute := TRUE;
    bResetRequested := TRUE;
END_IF

// Reset errors on the axis and motion FBs
IF bResetRequested THEN
    fbReset(Axis := Axis, Execute := bResetExecute);

    stStatus.bError := fbReset.Error;
    stStatus.iErrorCode := fbReset.ErrorID;

    IF fbReset.Error THEN
        stStatus.eState := E_ActuatorState.eError;
        stStatus.sMessage := 'Error in Reset';
        Reset := FALSE;
    ELSE
        stStatus.bError := FALSE;
        stStatus.iErrorCode := 0;
        stStatus.eState := E_ActuatorState.eIdle;
        stStatus.sMessage := '';
    END_IF;
	
	IF bResetDone THEN
        // Flags clearing  
        bResetRequested := FALSE;
        bResetDone := FALSE;
        Reset := TRUE;
        RETURN;
    END_IF
	
    IF fbReset.Done THEN
        bResetExecute := FALSE;
        bResetDone := TRUE;
    END_IF
    
END_IF

// Default Return
Reset := FALSE;
*)
END_METHOD

